C09106=1065.151,284.047,405.549,173.667,32.437,155.965
C09107=1065.146,283.799,405.580,173.664,32.433,155.964
C09108=1065.139,283.550,405.610,173.661,32.429,155.964
C09109=1065.133,283.302,405.641,173.659,32.425,155.963
C09110=1065.128,283.055,405.671,173.656,32.421,155.962
C09111=1065.121,282.806,405.702,173.653,32.416,155.961
C09112=1065.115,282.558,405.731,173.651,32.413,155.961
C09113=1065.109,282.311,405.762,173.648,32.409,155.960
C09114=1065.102,282.062,405.792,173.645,32.405,155.959
C09115=1065.097,281.814,405.823,173.642,32.401,155.958
C09116=1065.091,281.566,405.853,173.639,32.396,155.958
C09117=1065.084,281.318,405.884,173.637,32.393,155.957
C09118=1065.079,281.070,405.914,173.634,32.388,155.956
C09119=1065.073,280.822,405.945,173.631,32.384,155.955
C09120=1065.066,280.574,405.975,173.628,32.380,155.955
C09121=1065.060,280.326,406.006,173.625,32.376,155.954
C09122=1065.055,280.078,406.036,173.623,32.372,155.953
C09123=1065.048,279.829,406.065,173.621,32.368,155.952
C09124=1065.042,279.582,406.096,173.618,32.364,155.952
C09125=1065.036,279.334,406.126,173.615,32.360,155.951
C09126=1065.030,279.085,406.157,173.612,32.356,155.950
C09127=1065.023,278.838,406.187,173.609,32.352,155.949
C09128=1065.018,278.589,406.216,173.607,32.348,155.949
C09129=1065.011,278.341,406.247,173.604,32.344,155.948
C09130=1065.005,278.093,406.277,173.601,32.340,155.947
C09131=1064.999,277.845,406.306,173.598,32.336,155.946
C09132=1064.993,277.597,406.337,173.595,32.332,155.946
C09133=1064.987,277.377,406.364,173.594,32.328,155.945
C09134=1064.982,277.156,406.390,173.591,32.325,155.944
C09135=1064.976,276.936,406.417,173.589,32.321,155.944
C09136=1064.971,276.716,406.443,173.586,32.318,155.943
C09137=1064.966,276.496,406.470,173.584,32.314,155.942
C09138=1064.960,276.275,406.496,173.582,32.310,155.942
C09139=1064.955,276.055,406.524,173.579,32.307,155.941
C09140=1064.950,275.835,406.550,173.577,32.304,155.940
C09141=1064.943,275.587,406.580,173.574,32.299,155.940
C09142=1064.937,275.339,406.610,173.571,32.296,155.939
C09143=1064.932,275.091,406.640,173.568,32.291,155.938
C09144=1064.925,274.843,406.669,173.566,32.288,155.937
C09145=1064.920,274.595,406.699,173.564,32.283,155.937
C09146=1064.913,274.346,406.730,173.561,32.280,155.936
C09147=1064.907,274.098,406.759,173.558,32.275,155.935
C09148=1064.901,273.850,406.789,173.555,32.272,155.934
C09149=1064.895,273.602,406.818,173.553,32.267,155.934
C09150=1064.889,273.354,406.849,173.550,32.264,155.933
C09151=1064.883,273.106,406.878,173.547,32.259,155.932
C09152=1064.876,272.857,406.908,173.545,32.256,155.932
C09153=1064.870,272.609,406.937,173.542,32.251,155.931
C09154=1064.865,272.361,406.967,173.539,32.248,155.930
C09155=1064.858,272.113,406.997,173.537,32.243,155.929
C09156=1064.853,271.865,407.026,173.535,32.240,155.929
C09157=1064.846,271.617,407.055,173.532,32.235,155.928
C09158=1064.840,271.368,407.086,173.529,32.232,155.927
C09159=1064.834,271.120,407.115,173.526,32.227,155.926
C09160=1064.828,270.872,407.145,173.524,32.224,155.926
C09161=1064.822,270.624,407.175,173.521,32.219,155.925
C09162=1064.816,270.376,407.204,173.518,32.216,155.924
C09163=1064.810,270.128,407.233,173.515,32.211,155.923
C09164=1064.804,269.879,407.262,173.513,32.208,155.923
C09165=1064.798,269.632,407.293,173.511,32.204,155.922
C09166=1064.792,269.384,407.322,173.508,32.200,155.921
C09167=1064.786,269.135,407.351,173.506,32.196,155.921
C09168=1064.779,268.886,407.381,173.503,32.192,155.920
C09169=1064.773,268.639,407.410,173.500,32.188,155.919
C09170=1064.767,268.390,407.440,173.497,32.184,155.918
C09171=1064.761,268.142,407.469,173.495,32.180,155.918
C09172=1064.755,267.894,407.498,173.492,32.176,155.917
C09173=1064.749,267.646,407.528,173.489,32.172,155.916
C09174=1064.743,267.397,407.557,173.488,32.168,155.915
C09175=1064.737,267.149,407.586,173.485,32.164,155.915
C09176=1064.730,266.901,407.615,173.482,32.160,155.914
C09177=1064.725,266.653,407.645,173.480,32.156,155.913
C09178=1064.719,266.405,407.674,173.477,32.152,155.912
C09179=1064.712,266.157,407.703,173.474,32.148,155.912
C09180=1064.706,265.909,407.733,173.472,32.144,155.911
C09181=1064.700,265.661,407.762,173.469,32.140,155.910
C09182=1064.694,265.412,407.791,173.466,32.136,155.910
C09183=1064.688,265.164,407.820,173.465,32.133,155.909
C09184=1064.682,264.916,407.850,173.462,32.128,155.908
C09185=1064.676,264.667,407.878,173.459,32.124,155.907
C09186=1064.670,264.419,407.907,173.457,32.120,155.907
C09187=1064.664,264.171,407.936,173.454,32.116,155.906
C09188=1064.658,263.922,407.966,173.451,32.113,155.905
C09189=1064.653,263.704,407.991,173.449,32.109,155.905
C09190=1064.647,263.486,408.017,173.447,32.105,155.904
C09191=1064.642,263.268,408.042,173.444,32.102,155.903
C09192=1064.636,263.049,408.068,173.443,32.099,155.903
C09193=1064.631,262.831,408.093,173.440,32.095,155.902
C09194=1064.625,262.612,408.119,173.438,32.092,155.901
C09195=1064.619,262.393,408.144,173.436,32.089,155.901
C09196=1064.614,262.175,408.170,173.433,32.085,155.900
C09197=1064.608,261.927,408.199,173.431,32.081,155.899
C09198=1064.602,261.678,408.227,173.428,32.077,155.899
C09199=1064.595,261.430,408.256,173.425,32.073,155.898
C09200=1064.589,261.182,408.285,173.423,32.069,155.897
C09201=1064.583,260.934,408.314,173.421,32.066,155.897
C09202=1064.577,260.685,408.342,173.419,32.061,155.896
C09203=1064.571,260.437,408.371,173.416,32.058,155.895
C09204=1064.564,260.189,408.400,173.413,32.054,155.895
C09205=1064.558,259.940,408.429,173.411,32.050,155.894
C09206=1064.552,259.693,408.457,173.408,32.046,155.893
C09207=1064.546,259.445,408.486,173.405,32.042,155.892
C09208=1064.540,259.196,408.514,173.403,32.039,155.892
C09209=1064.534,258.948,408.543,173.401,32.034,155.891
C09210=1064.527,258.700,408.572,173.399,32.031,155.890
C09211=1064.521,258.451,408.601,173.396,32.027,155.890
C09212=1064.515,258.203,408.630,173.393,32.022,155.889
C09213=1064.509,257.954,408.658,173.391,32.019,155.888
C09214=1064.503,257.706,408.687,173.388,32.015,155.887
C09215=1064.496,257.458,408.715,173.385,32.011,155.887
C09216=1064.490,257.209,408.744,173.383,32.007,155.886
C09217=1064.485,256.961,408.772,173.381,32.003,155.885
C09218=1064.478,256.713,408.801,173.379,31.999,155.884
C09219=1064.473,256.464,408.829,173.376,31.995,155.884
C09220=1064.466,256.216,408.858,173.373,31.991,155.883
C09221=1064.460,255.968,408.886,173.371,31.987,155.882
C09222=1064.453,255.720,408.915,173.368,31.983,155.882
C09223=1064.448,255.472,408.943,173.366,31.979,155.881
C09224=1064.442,255.224,408.972,173.364,31.975,155.880
C09225=1064.436,254.975,409.000,173.362,31.972,155.880
C09226=1064.430,254.727,409.029,173.359,31.967,155.879
C09227=1064.424,254.478,409.058,173.356,31.964,155.878
C09228=1064.418,254.230,409.086,173.354,31.960,155.877
C09229=1064.411,253.982,409.114,173.351,31.956,155.877
C09230=1064.405,253.733,409.142,173.349,31.952,155.876
C09231=1064.399,253.485,409.171,173.347,31.948,155.875
C09232=1064.394,253.237,409.199,173.345,31.944,155.874
C09233=1064.388,252.988,409.228,173.342,31.940,155.874
C09234=1064.381,252.740,409.255,173.339,31.936,155.873
C09235=1064.375,252.492,409.284,173.337,31.932,155.872
C09236=1064.370,252.244,409.312,173.334,31.928,155.872
C09237=1064.364,251.995,409.341,173.332,31.924,155.871
C09238=1064.358,251.746,409.369,173.329,31.920,155.870
C09239=1064.351,251.498,409.397,173.328,31.916,155.869
C09240=1064.345,251.250,409.425,173.325,31.912,155.869
C09241=1064.339,251.002,409.454,173.323,31.908,155.868
C09242=1064.333,250.753,409.482,173.320,31.904,155.867
C09243=1064.328,250.505,409.510,173.318,31.901,155.867
C09244=1064.321,250.257,409.538,173.315,31.896,155.866
C09245=1064.316,250.037,409.564,173.313,31.893,155.865
C09246=1064.311,249.818,409.588,173.312,31.889,155.865
C09247=1064.305,249.598,409.613,173.309,31.886,155.864
C09248=1064.300,249.379,409.638,173.307,31.882,155.863
C09249=1064.295,249.159,409.663,173.305,31.879,155.863
C09250=1064.290,248.940,409.688,173.303,31.875,155.862
C09251=1064.285,248.720,409.713,173.300,31.871,155.861
C09252=1064.279,248.501,409.737,173.298,31.868,155.861
C09253=1064.273,248.252,409.766,173.297,31.864,155.860
C09254=1064.268,248.004,409.794,173.294,31.860,155.859
C09255=1064.261,247.755,409.821,173.292,31.856,155.858
C09256=1064.256,247.507,409.850,173.289,31.852,155.858
C09257=1064.250,247.259,409.878,173.287,31.848,155.857
C09258=1064.244,247.010,409.906,173.284,31.844,155.856
C09259=1064.238,246.762,409.933,173.282,31.840,155.856
C09260=1064.232,246.513,409.962,173.280,31.836,155.855
C09261=1064.227,246.265,409.990,173.278,31.832,155.854
C09262=1064.220,246.017,410.017,173.275,31.828,155.853
C09263=1064.214,245.768,410.046,173.273,31.824,155.853
C09264=1064.208,245.520,410.073,173.270,31.820,155.852
C09265=1064.202,245.272,410.101,173.268,31.816,155.851
C09266=1064.196,245.023,410.128,173.266,31.812,155.850
C09267=1064.190,244.775,410.156,173.264,31.808,155.850
C09268=1064.184,244.526,410.184,173.261,31.805,155.849
C09269=1064.178,244.278,410.212,173.259,31.800,155.848
C09270=1064.172,244.030,410.240,173.256,31.797,155.848
C09271=1064.166,243.782,410.268,173.254,31.792,155.847
C09272=1064.160,243.532,410.295,173.252,31.788,155.846
C09273=1064.154,243.284,410.323,173.250,31.785,155.846
C09274=1064.148,243.036,410.350,173.248,31.781,155.845
C09275=1064.142,242.787,410.379,173.245,31.777,155.844
C09276=1064.136,242.540,410.406,173.243,31.773,155.843
C09277=1064.130,242.290,410.434,173.240,31.769,155.843
C09278=1064.124,242.042,410.461,173.238,31.765,155.842
C09279=1064.118,241.794,410.489,173.236,31.761,155.841
C09280=1064.113,241.545,410.516,173.234,31.757,155.841
C09281=1064.106,241.297,410.544,173.231,31.753,155.840
C09282=1064.099,241.048,410.571,173.229,31.749,155.839
C09283=1064.094,240.800,410.599,173.226,31.745,155.838
C09284=1064.088,240.551,410.626,173.224,31.741,155.838
C09285=1064.081,240.304,410.654,173.223,31.737,155.837
C09286=1064.075,240.054,410.681,173.220,31.733,155.836
C09287=1064.070,239.806,410.709,173.218,31.730,155.836
C09288=1064.063,239.557,410.736,173.215,31.725,155.835
C09289=1064.057,239.310,410.763,173.213,31.722,155.834
C09290=1064.051,239.061,410.791,173.210,31.718,155.833
C09291=1064.046,238.813,410.818,173.209,31.714,155.833
C09292=1064.039,238.564,410.846,173.206,31.710,155.832
C09293=1064.033,238.316,410.873,173.204,31.705,155.831
C09294=1064.026,238.067,410.900,173.202,31.702,155.831
C09295=1064.021,237.819,410.928,173.199,31.698,155.830
C09296=1064.015,237.570,410.955,173.197,31.694,155.829
C09297=1064.009,237.322,410.982,173.195,31.690,155.828
C09298=1064.002,237.073,411.010,173.193,31.686,155.828
C09299=1063.996,236.825,411.036,173.190,31.682,155.827
C09300=1063.991,236.576,411.064,173.188,31.678,155.826
C09301=1063.985,236.354,411.088,173.186,31.674,155.826
C09302=1063.980,236.131,411.112,173.184,31.671,155.825
C09303=1063.975,235.909,411.137,173.183,31.668,155.824
C09304=1063.969,235.686,411.161,173.180,31.664,155.824
C09305=1063.964,235.463,411.186,173.178,31.660,155.823
C09306=1063.958,235.241,411.210,173.176,31.656,155.822
C09307=1063.953,235.018,411.234,173.174,31.653,155.822
C09308=1063.947,234.795,411.258,173.172,31.650,155.821
C09309=1063.941,234.547,411.286,173.170,31.646,155.820
C09310=1063.936,234.299,411.312,173.168,31.642,155.820
C09311=1063.929,234.049,411.339,173.166,31.638,155.819
C09312=1063.924,233.801,411.367,173.163,31.633,155.818
C09313=1063.918,233.553,411.394,173.161,31.630,155.818
C09314=1063.912,233.304,411.421,173.159,31.626,155.817
C09315=1063.906,233.056,411.448,173.157,31.622,155.816
C09316=1063.899,232.807,411.475,173.155,31.618,155.815
C09317=1063.893,232.559,411.502,173.152,31.614,155.815
C09318=1063.888,232.310,411.529,173.150,31.610,155.814
C09319=1063.881,232.061,411.556,173.148,31.606,155.813
C09320=1063.876,231.813,411.582,173.146,31.602,155.813
C09321=1063.869,231.565,411.610,173.144,31.598,155.812
C09322=1063.863,231.316,411.637,173.142,31.594,155.811
C09323=1063.857,231.068,411.663,173.139,31.590,155.810
C09324=1063.852,230.820,411.690,173.137,31.586,155.810
C09325=1063.845,230.570,411.717,173.135,31.582,155.809
C09326=1063.839,230.322,411.744,173.133,31.578,155.808
C09327=1063.833,230.074,411.771,173.131,31.574,155.807
C09328=1063.827,229.825,411.798,173.128,31.570,155.807
C09329=1063.821,229.577,411.825,173.126,31.566,155.806
C09330=1063.815,229.329,411.851,173.124,31.562,155.805
C09331=1063.809,229.080,411.878,173.122,31.558,155.805
C09332=1063.803,228.831,411.905,173.120,31.554,155.804
C09333=1063.797,228.583,411.932,173.118,31.550,155.803
C09334=1063.790,228.334,411.958,173.115,31.546,155.802
C09335=1063.785,228.086,411.985,173.113,31.542,155.802
C09336=1063.779,227.837,412.011,173.112,31.538,155.801
C09337=1063.773,227.589,412.038,173.109,31.534,155.800
C09338=1063.767,227.340,412.065,173.107,31.530,155.800
C09339=1063.760,227.092,412.091,173.105,31.526,155.799
C09340=1063.754,226.844,412.118,173.102,31.522,155.798
C09341=1063.748,226.594,412.144,173.101,31.518,155.797
C09342=1063.743,226.345,412.171,173.099,31.514,155.797
C09343=1063.737,226.097,412.197,173.096,31.510,155.796
C09344=1063.730,225.849,412.223,173.094,31.506,155.795
C09345=1063.724,225.600,412.251,173.092,31.503,155.795
C09346=1063.718,225.352,412.277,173.090,31.498,155.794
C09347=1063.712,225.103,412.304,173.088,31.494,155.793
C09348=1063.706,224.855,412.330,173.086,31.490,155.792
C09349=1063.700,224.606,412.356,173.083,31.486,155.792
C09350=1063.694,224.357,412.383,173.081,31.483,155.791
C09351=1063.688,224.109,412.409,173.080,31.478,155.790
C09352=1063.682,223.861,412.436,173.077,31.474,155.790
C09353=1063.676,223.612,412.462,173.075,31.470,155.789
C09354=1063.670,223.363,412.488,173.073,31.466,155.788
C09355=1063.664,223.114,412.515,173.071,31.462,155.787
C09356=1063.658,222.866,412.541,173.069,31.458,155.787
C09357=1063.652,222.640,412.565,173.067,31.455,155.786
C09358=1063.647,222.413,412.589,173.065,31.451,155.785
C09359=1063.642,222.186,412.614,173.063,31.447,155.785
C09360=1063.636,221.960,412.638,173.061,31.444,155.784
C09361=1063.631,221.733,412.662,173.059,31.440,155.783
C09362=1063.625,221.507,412.685,173.058,31.436,155.783
C09363=1063.620,221.280,412.709,173.056,31.432,155.782
C09364=1063.614,221.053,412.733,173.054,31.429,155.781
C09365=1063.608,220.805,412.759,173.051,31.425,155.781
C09366=1063.602,220.556,412.785,173.049,31.421,155.780
C09367=1063.597,220.308,412.812,173.048,31.417,155.779
C09368=1063.590,220.058,412.838,173.045,31.413,155.779
C09369=1063.584,219.810,412.864,173.043,31.409,155.778
C09370=1063.578,219.562,412.890,173.041,31.405,155.777
C09371=1063.572,219.313,412.916,173.040,31.401,155.776
C09372=1063.566,219.065,412.942,173.037,31.397,155.776
C09373=1063.560,218.816,412.968,173.035,31.393,155.775
C09374=1063.554,218.568,412.994,173.033,31.389,155.774
C09375=1063.548,218.319,413.020,173.031,31.385,155.773
C09376=1063.541,218.070,413.047,173.029,31.381,155.773
C09377=1063.536,217.821,413.073,173.027,31.377,155.772
C09378=1063.529,217.573,413.099,173.025,31.373,155.771
C09379=1063.523,217.324,413.124,173.023,31.369,155.771
C09380=1063.517,217.076,413.151,173.020,31.365,155.770
C09381=1063.511,216.827,413.176,173.019,31.361,155.769
C09382=1063.505,216.579,413.203,173.017,31.357,155.768
C09383=1063.499,216.330,413.228,173.015,31.353,155.768
C09384=1063.493,216.081,413.254,173.012,31.348,155.767
C09385=1063.487,215.833,413.280,173.011,31.345,155.766
C09386=1063.481,215.584,413.306,173.009,31.340,155.766
C09387=1063.475,215.336,413.332,173.007,31.337,155.765
C09388=1063.469,215.087,413.358,173.004,31.332,155.764
C09389=1063.463,214.839,413.383,173.002,31.328,155.763
C09390=1063.457,214.590,413.410,173.001,31.324,155.763
C09391=1063.451,214.342,413.435,172.999,31.320,155.762
C09392=1063.445,214.093,413.461,172.996,31.316,155.761
C09393=1063.439,213.845,413.487,172.994,31.312,155.760
C09394=1063.433,213.596,413.513,172.993,31.308,155.760
C09395=1063.428,213.347,413.539,172.991,31.304,155.759
C09396=1063.421,213.099,413.565,172.989,31.300,155.758
C09397=1063.416,212.850,413.591,172.986,31.296,155.757
C09398=1063.409,212.601,413.616,172.984,31.291,155.757
C09399=1063.403,212.352,413.641,172.983,31.288,155.756
C09400=1063.397,212.104,413.668,172.981,31.283,155.755
C09401=1063.391,211.855,413.693,172.979,31.280,155.755
C09402=1063.385,211.607,413.719,172.976,31.275,155.754
C09403=1063.379,211.358,413.744,172.975,31.271,155.753
C09404=1063.373,211.109,413.770,172.973,31.267,155.752
C09405=1063.367,210.860,413.795,172.971,31.263,155.752
C09406=1063.361,210.612,413.821,172.969,31.259,155.751
C09407=1063.354,210.364,413.847,172.967,31.255,155.750
C09408=1063.349,210.115,413.872,172.965,31.251,155.749
C09409=1063.343,209.866,413.898,172.963,31.247,155.749
C09410=1063.337,209.617,413.923,172.961,31.243,155.748
C09411=1063.330,209.369,413.949,172.959,31.239,155.747
C09412=1063.325,209.120,413.974,172.957,31.235,155.747
C09413=1063.319,208.896,413.997,172.955,31.231,155.746
C09414=1063.314,208.672,414.020,172.953,31.227,155.745
C09415=1063.308,208.448,414.044,172.951,31.224,155.745
C09416=1063.302,208.223,414.066,172.950,31.220,155.744
C09417=1063.298,207.999,414.089,172.949,31.216,155.743
C09418=1063.292,207.775,414.112,172.947,31.213,155.743
C09419=1063.286,207.551,414.135,172.945,31.209,155.742
C09420=1063.281,207.326,414.158,172.943,31.205,155.741
C09421=1063.256,206.279,414.261,172.776,31.124,155.734
C09422=1063.250,206.030,414.286,172.774,31.121,155.734
C09423=1063.245,205.781,414.310,172.771,31.118,155.733
C09424=1063.238,205.533,414.335,172.769,31.114,155.733
C09425=1063.233,205.284,414.359,172.766,31.111,155.732
C09426=1063.227,205.035,414.384,172.765,31.108,155.732
C09427=1063.222,204.787,414.408,172.763,31.105,155.731
C09428=1063.216,204.538,414.434,172.760,31.102,155.731
C09429=1063.210,204.289,414.458,172.758,31.099,155.730
C09430=1063.204,204.040,414.482,172.755,31.095,155.730
C09431=1063.198,203.792,414.506,172.754,31.092,155.729
C09432=1063.192,203.542,414.531,172.751,31.089,155.729
C09433=1063.187,203.294,414.556,172.749,31.086,155.728
C09434=1063.181,203.045,414.580,172.746,31.082,155.727
C09435=1063.176,202.797,414.605,172.744,31.079,155.727
C09436=1063.169,202.548,414.629,172.743,31.076,155.726
C09437=1063.164,202.299,414.653,172.740,31.073,155.726
C09438=1063.158,202.050,414.677,172.738,31.070,155.725
C09439=1063.152,201.801,414.701,172.735,31.067,155.725
C09440=1063.146,201.554,414.726,172.734,31.063,155.724
C09441=1063.140,201.304,414.751,172.731,31.061,155.724
C09442=1063.134,201.056,414.774,172.729,31.057,155.723
C09443=1063.128,200.807,414.799,172.727,31.054,155.723
C09444=1063.122,200.558,414.823,172.724,31.051,155.722
C09445=1063.116,200.309,414.847,172.723,31.048,155.722
C09446=1063.110,200.061,414.871,172.720,31.045,155.721
C09447=1063.104,199.812,414.896,172.718,31.042,155.721
C09448=1063.098,199.563,414.919,172.715,31.039,155.720
C09449=1063.092,199.314,414.944,172.713,31.036,155.720
C09450=1063.086,199.066,414.968,172.712,31.033,155.719
C09451=1063.081,198.817,414.992,172.709,31.030,155.719
C09452=1063.075,198.568,415.016,172.707,31.027,155.718
C09453=1063.070,198.319,415.039,172.704,31.023,155.718
C09454=1063.063,198.070,415.063,172.702,31.020,155.717
C09455=1063.058,197.821,415.088,172.701,31.017,155.717
C09456=1063.051,197.572,415.112,172.698,31.014,155.716
C09457=1063.046,197.324,415.136,172.696,31.011,155.716
C09458=1063.040,197.075,415.160,172.693,31.008,155.715
C09459=1063.034,196.826,415.184,172.692,31.005,155.715
C09460=1063.028,196.578,415.208,172.690,31.002,155.714
C09461=1063.022,196.329,415.232,172.687,30.999,155.714
C09462=1063.016,196.080,415.255,172.685,30.996,155.713
C09463=1063.011,195.831,415.280,172.682,30.992,155.713
C09464=1063.005,195.583,415.303,172.681,30.990,155.713
C09465=1062.999,195.334,415.328,172.679,30.987,155.712
C09466=1062.993,195.085,415.352,172.676,30.983,155.711
C09467=1062.988,194.836,415.375,172.674,30.981,155.711
C09468=1062.981,194.587,415.399,172.672,30.977,155.710
C09469=1062.975,194.339,415.423,172.670,30.974,155.710
C09470=1062.970,194.090,415.447,172.668,30.971,155.710
C09471=1062.963,193.841,415.470,172.666,30.968,155.709
C09472=1062.958,193.592,415.495,172.663,30.965,155.708
C09473=1062.952,193.344,415.518,172.662,30.962,155.708
C09474=1062.946,193.095,415.543,172.659,30.959,155.708
C09475=1062.940,192.846,415.566,172.657,30.956,155.707
C09476=1062.935,192.597,415.590,172.655,30.953,155.707
C09477=1062.929,192.349,415.614,172.652,30.950,155.706
C09478=1062.923,192.099,415.637,172.651,30.947,155.706
C09479=1062.918,191.851,415.661,172.649,30.944,155.705
C09480=1062.911,191.602,415.685,172.646,30.941,155.705
C09481=1062.907,191.353,415.709,172.644,30.937,155.704
C09482=1062.899,191.070,415.736,172.642,30.934,155.704
C09483=1062.893,190.786,415.762,172.640,30.931,155.703
C09484=1062.887,190.504,415.790,172.637,30.927,155.702
C09485=1062.879,190.220,415.817,172.634,30.924,155.702
C09486=1062.874,189.971,415.840,172.633,30.920,155.701
C09487=1062.868,189.723,415.864,172.631,30.918,155.701
C09488=1062.863,189.474,415.887,172.629,30.914,155.700
C09489=1062.857,189.225,415.912,172.626,30.911,155.700
C09490=1062.851,188.976,415.934,172.624,30.908,155.699
C09491=1062.846,188.727,415.959,172.623,30.905,155.699
C09492=1062.840,188.478,415.982,172.620,30.902,155.698
C09493=1062.834,188.230,416.005,172.618,30.899,155.698
C09494=1062.829,187.981,416.029,172.616,30.896,155.697
C09495=1062.822,187.732,416.053,172.613,30.893,155.697
C09496=1062.817,187.483,416.076,172.612,30.890,155.696
C09497=1062.811,187.234,416.100,172.610,30.887,155.696
C09498=1062.806,186.986,416.123,172.608,30.884,155.695
C09499=1062.800,186.737,416.147,172.605,30.881,155.695
C09500=1062.795,186.488,416.170,172.604,30.878,155.694
C09501=1062.789,186.240,416.194,172.602,30.875,155.694
C09502=1062.784,185.991,416.217,172.599,30.872,155.694
C09503=1062.778,185.742,416.240,172.597,30.868,155.693
C09504=1062.771,185.493,416.264,172.595,30.866,155.693
C09505=1062.766,185.244,416.288,172.594,30.863,155.692
C09506=1062.760,184.995,416.312,172.591,30.859,155.691
C09507=1062.755,184.746,416.335,172.589,30.857,155.691
C09508=1062.749,184.497,416.358,172.587,30.853,155.691
C09509=1062.744,184.248,416.381,172.585,30.851,155.690
C09510=1062.738,184.000,416.405,172.583,30.847,155.690
C09511=1062.731,183.750,416.428,172.581,30.845,155.689
C09512=1062.725,183.502,416.450,172.579,30.842,155.689
C09513=1062.719,183.253,416.473,172.577,30.839,155.688
C09514=1062.713,183.005,416.497,172.575,30.836,155.688
C09515=1062.707,182.756,416.520,172.573,30.834,155.687
C09516=1062.701,182.506,416.543,172.570,30.830,155.687
C09517=1062.695,182.257,416.566,172.568,30.827,155.686
C09518=1062.690,182.008,416.589,172.567,30.825,155.686
C09519=1062.684,181.760,416.613,172.565,30.822,155.686
C09520=1062.678,181.511,416.636,172.562,30.819,155.685
C09521=1062.671,181.263,416.658,172.560,30.816,155.685
C09522=1062.665,181.013,416.681,172.558,30.813,155.684
C09523=1062.659,180.764,416.704,172.557,30.810,155.684
C09524=1062.654,180.515,416.727,172.554,30.808,155.683
C09525=1062.648,180.266,416.750,172.552,30.804,155.683
C09526=1062.642,180.018,416.774,172.550,30.802,155.682
C09527=1062.636,179.769,416.797,172.549,30.798,155.682
C09528=1062.630,179.520,416.820,172.546,30.796,155.681
C09529=1062.624,179.272,416.842,172.544,30.793,155.681
C09530=1062.618,179.023,416.865,172.542,30.790,155.680
C09531=1062.612,178.773,416.888,172.540,30.787,155.680
C09532=1062.606,178.524,416.911,172.538,30.784,155.680
C09533=1062.600,178.275,416.934,172.536,30.781,155.679
C09534=1062.595,178.026,416.957,172.534,30.779,155.679
C09535=1062.588,177.778,416.980,172.532,30.776,155.678
C09536=1062.582,177.529,417.003,172.530,30.772,155.678
C09537=1062.577,177.280,417.026,172.528,30.770,155.677
C09538=1062.571,177.031,417.048,172.526,30.767,155.677
C09539=1062.565,176.782,417.071,172.524,30.764,155.676
C09540=1062.559,176.533,417.094,172.521,30.761,155.676
C09541=1062.553,176.285,417.117,172.520,30.759,155.676
C09542=1062.547,176.036,417.140,172.518,30.755,155.675
C09543=1062.542,175.787,417.163,172.516,30.753,155.675
C09544=1062.536,175.538,417.186,172.514,30.749,155.674
C09545=1062.530,175.289,417.208,172.512,30.747,155.674
C09546=1062.524,175.005,417.234,172.510,30.743,155.673
C09547=1062.517,174.722,417.260,172.507,30.740,155.673
C09548=1062.510,174.439,417.286,172.505,30.737,155.672
C09549=1062.504,174.155,417.312,172.503,30.733,155.672
C09550=1062.498,173.906,417.334,172.501,30.731,155.671
C09551=1062.492,173.657,417.357,172.499,30.728,155.671
C09552=1062.486,173.408,417.380,172.497,30.725,155.670
C09553=1062.480,173.159,417.403,172.495,30.722,155.670
C09554=1062.475,172.910,417.425,172.493,30.719,155.669
C09555=1062.468,172.661,417.447,172.491,30.716,155.669
C09556=1062.462,172.412,417.470,172.489,30.714,155.668
C09557=1062.457,172.164,417.493,172.487,30.710,155.668
C09558=1062.451,171.915,417.516,172.486,30.708,155.668
C09559=1062.446,171.665,417.538,172.483,30.705,155.667
C09560=1062.439,171.417,417.561,172.481,30.702,155.667
C09561=1062.433,171.168,417.584,172.479,30.699,155.666
C09562=1062.428,170.919,417.607,172.478,30.696,155.666
C09563=1062.423,170.670,417.628,172.476,30.693,155.665
C09564=1062.416,170.421,417.651,172.474,30.691,155.665
C09565=1062.411,170.173,417.674,172.471,30.688,155.664
C09566=1062.405,169.924,417.697,172.469,30.684,155.664
C09567=1062.399,169.674,417.719,172.468,30.682,155.663
C09568=1062.393,169.426,417.741,172.466,30.679,155.663
C09569=1062.387,169.177,417.764,172.464,30.676,155.662
C09570=1062.382,168.928,417.786,172.462,30.673,155.662
C09571=1062.377,168.679,417.809,172.460,30.670,155.662
C09572=1062.370,168.430,417.831,172.458,30.667,155.661
C09573=1062.365,168.181,417.854,172.456,30.665,155.661
C09574=1062.359,167.932,417.877,172.454,30.661,155.660
C09575=1062.353,167.683,417.898,172.453,30.659,155.660
C09576=1062.348,167.435,417.921,172.451,30.656,155.659
C09577=1062.342,167.186,417.944,172.449,30.653,155.659
C09578=1062.337,166.936,417.966,172.446,30.650,155.658
C09579=1062.330,166.688,417.988,172.444,30.647,155.658
C09580=1062.325,166.438,418.011,172.443,30.644,155.657
C09581=1062.320,166.190,418.033,172.441,30.642,155.657
C09582=1062.313,165.941,418.055,172.439,30.638,155.657
C09583=1062.308,165.692,418.078,172.437,30.636,155.656
C09584=1062.302,165.443,418.101,172.436,30.633,155.656
C09585=1062.297,165.193,418.123,172.434,30.630,155.655
C09586=1062.291,164.945,418.145,172.431,30.627,155.655
C09587=1062.285,164.696,418.167,172.429,30.624,155.654
C09588=1062.280,164.447,418.190,172.428,30.621,155.654
C09589=1062.273,164.198,418.212,172.426,30.618,155.653
C09590=1062.268,163.950,418.234,172.424,30.615,155.653
C09591=1062.263,163.700,418.256,172.422,30.612,155.652
C09592=1062.257,163.451,418.278,172.420,30.610,155.652
C09593=1062.251,163.202,418.301,172.419,30.607,155.652
C09594=1062.246,162.953,418.323,172.417,30.604,155.651
C09595=1062.240,162.705,418.345,172.414,30.601,155.651
C09596=1062.234,162.455,418.368,172.412,30.598,155.650
C09597=1062.229,162.207,418.390,172.411,30.595,155.650
C09598=1062.223,161.958,418.412,172.409,30.592,155.649
C09599=1062.217,161.708,418.434,172.407,30.589,155.649
C09600=1062.212,161.460,418.457,172.405,30.586,155.648
C09601=1062.206,161.211,418.478,172.404,30.583,155.648
C09602=1062.201,160.961,418.500,172.402,30.581,155.647
C09603=1062.194,160.713,418.523,172.400,30.578,155.647
C09604=1062.189,160.464,418.544,172.398,30.575,155.646
C09605=1062.183,160.215,418.566,172.396,30.572,155.646
C09606=1062.177,159.966,418.589,172.394,30.569,155.646
C09607=1062.171,159.717,418.610,172.392,30.567,155.645
C09608=1062.166,159.468,418.632,172.390,30.564,155.645
C09609=1062.160,159.219,418.654,172.388,30.561,155.644
C09610=1062.153,158.935,418.679,172.387,30.558,155.644
C09611=1062.146,158.651,418.704,172.384,30.555,155.643
C09612=1062.140,158.367,418.729,172.382,30.552,155.643
C09613=1062.133,158.083,418.753,172.381,30.548,155.642
C09614=1062.127,157.834,418.776,172.378,30.545,155.642
C09615=1062.121,157.585,418.798,172.376,30.543,155.642
C09616=1062.115,157.337,418.819,172.374,30.540,155.641
C09617=1062.110,157.087,418.842,172.373,30.537,155.641
C09618=1062.104,156.838,418.863,172.371,30.534,155.640
C09619=1062.098,156.589,418.884,172.369,30.532,155.640
C09620=1062.092,156.340,418.907,172.367,30.529,155.639
C09621=1062.086,156.091,418.929,172.365,30.526,155.639
C09622=1062.081,155.843,418.950,172.364,30.523,155.638
C09623=1062.075,155.593,418.972,172.362,30.520,155.638
C09624=1062.069,155.344,418.994,172.360,30.518,155.638
C09625=1062.064,155.095,419.015,172.358,30.515,155.637
C09626=1062.057,154.846,419.037,172.357,30.512,155.637
C09627=1062.051,154.597,419.059,172.354,30.510,155.636
C09628=1062.046,154.349,419.080,172.352,30.506,155.636
C09629=1062.040,154.099,419.102,172.350,30.504,155.635
C09630=1062.034,153.850,419.124,172.349,30.501,155.635
C09631=1062.029,153.601,419.145,172.347,30.498,155.635
C09632=1062.022,153.352,419.167,172.345,30.496,155.634
C09633=1062.016,153.103,419.188,172.343,30.493,155.634
C09634=1062.010,152.855,419.210,172.342,30.490,155.633
C09635=1062.005,152.605,419.232,172.340,30.487,155.633
C09636=1061.999,152.356,419.254,172.338,30.484,155.632
C09637=1061.994,152.107,419.275,172.336,30.482,155.632
C09638=1061.987,151.858,419.296,172.334,30.479,155.632
C09639=1061.982,151.609,419.318,172.333,30.476,155.631
C09640=1061.976,151.360,419.339,172.331,30.474,155.631
C09641=1061.969,151.111,419.361,172.329,30.470,155.630
C09642=1061.964,150.863,419.382,172.327,30.468,155.630
C09643=1061.958,150.613,419.404,172.326,30.465,155.629
C09644=1061.953,150.365,419.426,172.324,30.462,155.629
C09645=1061.947,150.115,419.447,172.322,30.460,155.629
C09646=1061.941,149.866,419.469,172.320,30.457,155.628
C09647=1061.935,149.618,419.490,172.319,30.454,155.628
C09648=1061.929,149.368,419.512,172.317,30.451,155.627
C09649=1061.924,149.119,419.532,172.314,30.448,155.627
C09650=1061.917,148.870,419.554,172.312,30.446,155.626
C09651=1061.912,148.622,419.575,172.311,30.443,155.626
C09652=1061.906,148.372,419.597,172.309,30.440,155.626
C09653=1061.900,148.123,419.619,172.307,30.438,155.625
C09654=1061.894,147.875,419.640,172.305,30.434,155.625
C09655=1061.888,147.625,419.661,172.304,30.432,155.624
C09656=1061.883,147.376,419.682,172.302,30.429,155.624
C09657=1061.876,147.127,419.704,172.300,30.426,155.623
C09658=1061.871,146.879,419.725,172.298,30.424,155.623
C09659=1061.865,146.629,419.746,172.296,30.421,155.623
C09660=1061.859,146.380,419.768,172.295,30.418,155.622
C09661=1061.853,146.131,419.789,172.293,30.416,155.622
C09662=1061.847,145.882,419.810,172.291,30.413,155.621
C09663=1061.842,145.633,419.831,172.289,30.410,155.621
C09664=1061.835,145.384,419.852,172.288,30.408,155.620
C09665=1061.829,145.135,419.873,172.286,30.405,155.620
C09666=1061.824,144.886,419.894,172.284,30.402,155.620
C09667=1061.818,144.637,419.916,172.282,30.399,155.619
C09668=1061.812,144.388,419.937,172.281,30.396,155.619
C09669=1061.806,144.139,419.958,172.279,30.394,155.618
C09670=1061.800,143.889,419.979,172.277,30.391,155.618
C09671=1061.795,143.641,420.001,172.275,30.388,155.617
C09672=1061.789,143.391,420.022,172.274,30.386,155.617
C09673=1061.783,143.143,420.042,172.272,30.383,155.617
C09674=1061.777,142.859,420.067,172.270,30.380,155.616
C09675=1061.769,142.574,420.091,172.268,30.377,155.616
C09676=1061.763,142.290,420.115,172.266,30.374,155.615
C09677=1061.756,142.006,420.139,172.264,30.370,155.615
C09678=1061.751,141.757,420.160,172.262,30.368,155.614
C09679=1061.745,141.507,420.181,172.260,30.365,155.614
C09680=1061.739,141.258,420.202,172.259,30.362,155.613
C09681=1061.732,141.009,420.223,172.257,30.360,155.613
C09682=1061.727,140.760,420.244,172.255,30.357,155.613
C09683=1061.721,140.511,420.265,172.253,30.354,155.612
C09684=1061.715,140.263,420.286,172.252,30.351,155.612
C09685=1061.710,140.013,420.307,172.250,30.348,155.611
C09686=1061.703,139.765,420.328,172.248,30.346,155.611
C09687=1061.698,139.515,420.349,172.246,30.343,155.610
C09688=1061.692,139.266,420.369,172.245,30.340,155.610
C09689=1061.687,139.017,420.391,172.243,30.338,155.610
C09690=1061.680,138.768,420.411,172.241,30.335,155.609
C09691=1061.674,138.519,420.432,172.239,30.332,155.609
C09692=1061.669,138.270,420.453,172.238,30.330,155.608
C09693=1061.662,138.021,420.474,172.236,30.327,155.608
C09694=1061.657,137.772,420.494,172.234,30.324,155.608
C09695=1061.651,137.523,420.516,172.232,30.322,155.607
C09696=1061.645,137.274,420.536,172.232,30.319,155.607
C09697=1061.639,137.024,420.557,172.230,30.316,155.606
C09698=1061.633,136.776,420.578,172.228,30.314,155.606
C09699=1061.627,136.527,420.598,172.226,30.311,155.605
C09700=1061.622,136.277,420.619,172.225,30.308,155.605
C09701=1061.616,136.028,420.640,172.223,30.306,155.605
C09702=1061.609,135.779,420.661,172.221,30.302,155.604
C09703=1061.604,135.530,420.682,172.219,30.300,155.604
C09704=1061.598,135.282,420.702,172.218,30.297,155.603
C09705=1061.592,135.032,420.723,172.216,30.294,155.603
C09706=1061.587,134.783,420.743,172.214,30.292,155.602
C09707=1061.580,134.534,420.764,172.212,30.289,155.602
C09708=1061.575,134.285,420.785,172.211,30.286,155.602
C09709=1061.569,134.035,420.806,172.209,30.284,155.601
C09710=1061.562,133.787,420.827,172.207,30.281,155.601
C09711=1061.557,133.537,420.847,172.205,30.278,155.600
C09712=1061.551,133.289,420.867,172.204,30.276,155.600
C09713=1061.545,133.039,420.888,172.202,30.273,155.600
C09714=1061.540,132.790,420.909,172.200,30.270,155.599
C09715=1061.534,132.542,420.929,172.198,30.268,155.599
C09716=1061.528,132.292,420.950,172.197,30.265,155.598
C09717=1061.522,132.043,420.970,172.196,30.262,155.598
C09718=1061.516,131.794,420.991,172.194,30.260,155.598
C09719=1061.510,131.545,421.012,172.192,30.257,155.597
C09720=1061.504,131.296,421.032,172.190,30.254,155.597
C09721=1061.498,131.047,421.052,172.189,30.252,155.596
C09722=1061.492,130.797,421.073,172.187,30.249,155.596
C09723=1061.487,130.548,421.093,172.185,30.246,155.595
C09724=1061.480,130.299,421.113,172.183,30.244,155.595
C09725=1061.474,130.051,421.134,172.182,30.241,155.595
C09726=1061.468,129.801,421.155,172.180,30.238,155.594
C09727=1061.462,129.552,421.175,172.178,30.235,155.594
C09728=1061.456,129.303,421.195,172.176,30.233,155.593
C09729=1061.451,129.054,421.216,172.175,30.230,155.593
C09730=1061.444,128.804,421.236,172.173,30.227,155.593
C09731=1061.438,128.556,421.256,172.171,30.225,155.592
C09732=1061.433,128.307,421.276,172.169,30.223,155.592
C09733=1061.426,128.057,421.297,172.169,30.220,155.591
C09734=1061.420,127.808,421.317,172.167,30.217,155.591
C09735=1061.415,127.559,421.337,172.165,30.215,155.591
C09736=1061.408,127.310,421.358,172.163,30.212,155.590
C09737=1061.402,127.061,421.378,172.162,30.209,155.590
C09738=1061.396,126.777,421.402,172.160,30.206,155.589
C09739=1061.389,126.492,421.424,172.157,30.203,155.589
C09740=1061.382,126.208,421.447,172.156,30.200,155.588
C09741=1061.375,125.923,421.470,172.154,30.197,155.588
C09742=1061.369,125.675,421.490,172.152,30.195,155.588
C09743=1061.364,125.425,421.511,172.150,30.192,155.587
C09744=1061.358,125.177,421.531,172.149,30.189,155.587
C09745=1061.351,124.927,421.551,172.147,30.186,155.586
C09746=1061.346,124.678,421.572,172.146,30.184,155.586
C09747=1061.340,124.429,421.591,172.144,30.181,155.586
C09748=1061.334,124.180,421.611,172.143,30.179,155.585
C09749=1061.327,123.931,421.632,172.141,30.176,155.585
C09750=1061.322,123.681,421.652,172.139,30.173,155.584
C09751=1061.316,123.432,421.672,172.137,30.170,155.584
C09752=1061.310,123.183,421.692,172.136,30.168,155.583
C09753=1061.305,122.934,421.712,172.134,30.165,155.583
C09754=1061.298,122.685,421.732,172.132,30.162,155.583
C09755=1061.292,122.436,421.752,172.130,30.160,155.582
C09756=1061.286,122.187,421.772,172.129,30.157,155.582
C09757=1061.281,121.938,421.793,172.128,30.155,155.581
C09758=1061.276,121.689,421.812,172.126,30.152,155.581
C09759=1061.269,121.439,421.832,172.124,30.149,155.581
C09760=1061.263,121.190,421.852,172.123,30.146,155.580
C09761=1061.258,120.941,421.873,172.121,30.144,155.580
C09762=1061.252,120.692,421.893,172.119,30.141,155.579
C09763=1061.246,120.443,421.912,172.117,30.138,155.579
C09764=1061.240,120.194,421.932,172.116,30.136,155.579
C09765=1061.234,119.944,421.953,172.115,30.133,155.578
C09766=1061.228,119.695,421.973,172.113,30.130,155.578
C09767=1061.222,119.446,421.992,172.111,30.128,155.577
C09768=1061.217,119.197,422.012,172.110,30.125,155.577
C09769=1061.211,118.948,422.032,172.108,30.122,155.576
C09770=1061.205,118.699,422.053,172.106,30.120,155.576
C09771=1061.200,118.450,422.072,172.105,30.117,155.576
C09772=1061.194,118.201,422.092,172.103,30.114,155.575
C09773=1061.187,117.952,422.112,172.101,30.112,155.575
C09774=1061.182,117.702,422.133,172.100,30.109,155.574
C09775=1061.176,117.453,422.152,172.099,30.106,155.574
C09776=1061.170,117.204,422.172,172.097,30.104,155.574
C09777=1061.164,116.955,422.192,172.095,30.101,155.573
C09778=1061.158,116.706,422.211,172.093,30.098,155.573
C09779=1061.153,116.457,422.232,172.092,30.096,155.572
C09780=1061.147,116.208,422.252,172.090,30.093,155.572
C09781=1061.141,115.959,422.271,172.089,30.090,155.572
C09782=1061.135,115.710,422.291,172.087,30.088,155.571
C09783=1061.130,115.460,422.310,172.086,30.084,155.571
C09784=1061.124,115.211,422.331,172.084,30.082,155.570
C09785=1061.118,114.962,422.351,172.082,30.079,155.570
C09786=1061.112,114.712,422.370,172.080,30.076,155.569
C09787=1061.106,114.463,422.390,172.079,30.074,155.569
C09788=1061.101,114.214,422.409,172.078,30.071,155.569
C09789=1061.095,113.965,422.429,172.076,30.068,155.568
C09790=1061.089,113.716,422.449,172.074,30.066,155.568
C09791=1061.083,113.467,422.469,172.073,30.063,155.567
C09792=1061.077,113.218,422.489,172.071,30.060,155.567
C09793=1061.071,112.969,422.508,172.069,30.057,155.566
C09794=1061.065,112.720,422.528,172.068,30.055,155.566
C09795=1061.059,112.470,422.547,172.067,30.053,155.566
C09796=1061.053,112.222,422.567,172.065,30.050,155.565
C09797=1061.048,111.972,422.586,172.063,30.047,155.565
C09798=1061.042,111.723,422.606,172.062,30.045,155.565
C09799=1061.036,111.474,422.625,172.060,30.042,155.564
C09800=1061.030,111.224,422.645,172.058,30.039,155.564
C09801=1061.024,110.975,422.665,172.056,30.037,155.563
C09802=1061.018,110.691,422.687,172.055,30.033,155.563
C09803=1061.010,110.406,422.709,172.053,30.031,155.562
C09804=1061.004,110.121,422.731,172.051,30.028,155.562
C09805=1060.997,109.838,422.754,172.050,30.025,155.561
C09806=1060.990,109.588,422.773,172.048,30.022,155.561
C09807=1060.984,109.339,422.793,172.046,30.019,155.561
C09808=1060.978,109.090,422.812,172.044,30.016,155.560
C09809=1060.973,108.840,422.831,172.043,30.014,155.560
C09810=1060.967,108.591,422.851,172.042,30.012,155.560
C09811=1060.961,108.342,422.870,172.040,30.009,155.559
C09812=1060.955,108.093,422.889,172.038,30.006,155.559
C09813=1060.949,107.844,422.909,172.037,30.004,155.558
C09814=1060.943,107.595,422.928,172.035,30.001,155.558
C09815=1060.937,107.345,422.947,172.033,29.998,155.558
C09816=1060.931,107.096,422.967,172.032,29.996,155.557
C09817=1060.925,106.847,422.986,172.031,29.993,155.557
C09818=1060.919,106.598,423.005,172.029,29.990,155.556
C09819=1060.913,106.349,423.025,172.027,29.988,155.556
C09820=1060.907,106.100,423.044,172.025,29.986,155.556
C09821=1060.901,105.850,423.063,172.024,29.983,155.555
C09822=1060.895,105.601,423.082,172.022,29.980,155.555
C09823=1060.889,105.352,423.102,172.021,29.978,155.554
C09824=1060.884,105.103,423.122,172.020,29.975,155.554
C09825=1060.878,104.853,423.141,172.018,29.972,155.554
C09826=1060.871,104.604,423.159,172.016,29.969,155.553
C09827=1060.865,104.355,423.179,172.014,29.967,155.553
C09828=1060.860,104.107,423.198,172.013,29.964,155.552
C09829=1060.855,103.857,423.218,172.012,29.962,155.552
C09830=1060.848,103.608,423.236,172.010,29.959,155.551
C09831=1060.843,103.359,423.255,172.008,29.956,155.551
C09832=1060.837,103.110,423.275,172.007,29.953,155.551
C09833=1060.831,102.860,423.295,172.005,29.951,155.550
C09834=1060.824,102.611,423.313,172.004,29.948,155.550
C09835=1060.819,102.362,423.333,172.003,29.945,155.549
C09836=1060.813,102.112,423.352,172.001,29.943,155.549
C09837=1060.807,101.863,423.371,171.999,29.940,155.549
C09838=1060.801,101.614,423.390,171.997,29.937,155.548
C09839=1060.795,101.365,423.410,171.996,29.935,155.548
C09840=1060.790,101.116,423.428,171.995,29.933,155.547
C09841=1060.784,100.867,423.448,171.993,29.930,155.547
C09842=1060.778,100.618,423.466,171.991,29.927,155.547
C09843=1060.772,100.368,423.486,171.990,29.924,155.546
C09844=1060.766,100.119,423.504,171.988,29.922,155.546
C09845=1060.760,99.870,423.524,171.986,29.919,155.545
C09846=1060.754,99.621,423.542,171.985,29.917,155.545
C09847=1060.748,99.371,423.561,171.984,29.914,155.545
C09848=1060.741,99.122,423.580,171.982,29.912,155.544
C09849=1060.736,98.873,423.599,171.980,29.909,155.544
C09850=1060.729,98.624,423.618,171.979,29.906,155.544
C09851=1060.724,98.374,423.637,171.978,29.904,155.543
C09852=1060.717,98.125,423.656,171.976,29.901,155.543
C09853=1060.712,97.876,423.675,171.974,29.898,155.542
C09854=1060.706,97.627,423.693,171.973,29.896,155.542
C09855=1060.700,97.378,423.713,171.971,29.893,155.542
C09856=1060.694,97.129,423.731,171.969,29.891,155.541
C09857=1060.688,96.879,423.750,171.968,29.888,155.541
C09858=1060.682,96.630,423.769,171.967,29.885,155.540
C09859=1060.676,96.381,423.788,171.965,29.883,155.540
C09860=1060.669,96.131,423.807,171.963,29.880,155.540
C09861=1060.664,95.883,423.826,171.962,29.877,155.539
C09862=1060.658,95.634,423.845,171.961,29.875,155.539
C09863=1060.652,95.384,423.864,171.959,29.873,155.538
C09864=1060.646,95.135,423.882,171.957,29.870,155.538
C09865=1060.640,94.885,423.901,171.956,29.867,155.538
C09866=1060.633,94.601,423.922,171.954,29.864,155.537
C09867=1060.627,94.317,423.944,171.952,29.861,155.537
C09868=1060.620,94.032,423.965,171.951,29.858,155.536
C09869=1060.613,93.748,423.987,171.949,29.855,155.536
C09870=1060.607,93.499,424.005,171.947,29.852,155.535
C09871=1060.601,93.249,424.024,171.945,29.850,155.535
C09872=1060.595,93.000,424.043,171.944,29.847,155.535
C09873=1060.590,92.751,424.061,171.943,29.844,155.534
C09874=1060.584,92.502,424.080,171.941,29.842,155.534
C09875=1060.578,92.252,424.099,171.939,29.840,155.533
C09876=1060.571,92.003,424.118,171.938,29.837,155.533
C09877=1060.566,91.754,424.137,171.936,29.834,155.533
C09878=1060.560,91.505,424.155,171.935,29.832,155.532
C09879=1060.555,91.255,424.174,171.934,29.829,155.532
C09880=1060.548,91.006,424.193,171.932,29.826,155.531
C09881=1060.542,90.757,424.211,171.930,29.823,155.531
C09882=1060.537,90.508,424.229,171.928,29.821,155.531
C09883=1060.531,90.258,424.248,171.928,29.818,155.530
C09884=1060.524,90.009,424.267,171.926,29.816,155.530
C09885=1060.518,89.760,424.285,171.924,29.813,155.529
C09886=1060.512,89.510,424.304,171.923,29.811,155.529
C09887=1060.506,89.262,424.322,171.921,29.808,155.529
C09888=1060.500,89.013,424.341,171.920,29.805,155.528
C09889=1060.494,88.763,424.359,171.918,29.803,155.528
C09890=1060.488,88.513,424.378,171.917,29.800,155.528
C09891=1060.482,88.264,424.397,171.915,29.798,155.527
C09892=1060.476,88.015,424.414,171.913,29.795,155.527
C09893=1060.470,87.766,424.433,171.912,29.792,155.526
C09894=1060.463,87.517,424.451,171.911,29.790,155.526
C09895=1060.458,87.267,424.470,171.909,29.788,155.526
C09896=1060.452,87.019,424.488,171.907,29.785,155.525
C09897=1060.446,86.769,424.506,171.906,29.782,155.525
C09898=1060.440,86.520,424.525,171.905,29.780,155.524
C09899=1060.433,86.271,424.543,171.903,29.777,155.524
C09900=1060.428,86.021,424.562,171.901,29.774,155.524
C09901=1060.422,85.772,424.580,171.900,29.772,155.523
C09902=1060.416,85.522,424.598,171.898,29.769,155.523
C09903=1060.410,85.274,424.617,171.897,29.767,155.522
C09904=1060.404,85.024,424.634,171.895,29.764,155.522
C09905=1060.398,84.775,424.653,171.894,29.761,155.522
C09906=1060.392,84.526,424.672,171.892,29.759,155.521
C09907=1060.386,84.277,424.690,171.890,29.756,155.521
C09908=1060.380,84.027,424.709,171.890,29.754,155.521
C09909=1060.374,83.778,424.726,171.888,29.751,155.520
C09910=1060.368,83.529,424.745,171.886,29.748,155.520
C09911=1060.362,83.280,424.763,171.884,29.746,155.519
C09912=1060.356,83.030,424.782,171.884,29.743,155.519
C09913=1060.351,82.781,424.800,171.882,29.740,155.518
C09914=1060.344,82.532,424.818,171.880,29.738,155.518
C09915=1060.338,82.282,424.836,171.879,29.736,155.518
C09916=1060.333,82.033,424.854,171.877,29.733,155.517
C09917=1060.326,81.784,424.872,171.876,29.730,155.517
C09918=1060.321,81.534,424.891,171.874,29.728,155.517
C09919=1060.315,81.286,424.909,171.873,29.725,155.516
C09920=1060.309,81.036,424.927,171.871,29.722,155.516
C09921=1060.302,80.787,424.946,171.869,29.720,155.515
C09922=1060.297,80.538,424.963,171.869,29.717,155.515
C09923=1060.291,80.288,424.981,171.867,29.715,155.515
C09924=1060.285,80.040,424.999,171.865,29.712,155.514
C09925=1060.280,79.789,425.018,171.863,29.709,155.514
C09926=1060.273,79.540,425.037,171.863,29.707,155.513
C09927=1060.268,79.291,425.054,171.861,29.704,155.513
C09928=1060.262,79.042,425.072,171.859,29.701,155.513
C09929=1060.255,78.792,425.091,171.858,29.699,155.512
C09930=1060.248,78.508,425.111,171.856,29.696,155.512
C09931=1060.242,78.223,425.131,171.854,29.693,155.511
C09932=1060.235,77.939,425.152,171.853,29.690,155.511
C09933=1060.228,77.655,425.173,171.851,29.687,155.510
C09934=1060.222,77.405,425.191,171.849,29.684,155.510
C09935=1060.216,77.157,425.209,171.848,29.682,155.510
C09936=1060.210,76.907,425.227,171.847,29.680,155.509
C09937=1060.204,76.658,425.244,171.845,29.677,155.509
C09938=1060.198,76.408,425.262,171.843,29.674,155.509
C09939=1060.192,76.159,425.281,171.842,29.671,155.508
C09940=1060.186,75.910,425.298,171.841,29.669,155.508
C09941=1060.180,75.660,425.316,171.839,29.667,155.507
C09942=1060.173,75.411,425.334,171.837,29.664,155.507
C09943=1060.168,75.162,425.351,171.836,29.661,155.507
C09944=1060.162,74.913,425.370,171.834,29.658,155.506
C09945=1060.156,74.664,425.388,171.833,29.656,155.506
C09946=1060.150,74.414,425.406,171.831,29.654,155.506
C09947=1060.144,74.165,425.423,171.830,29.651,155.505
C09948=1060.138,73.915,425.441,171.828,29.648,155.505
C09949=1060.131,73.666,425.459,171.827,29.646,155.504
C09950=1060.126,73.417,425.477,171.826,29.644,155.504
C09951=1060.119,73.167,425.495,171.824,29.641,155.504
C09952=1060.114,72.918,425.512,171.822,29.638,155.503
C09953=1060.108,72.669,425.530,171.821,29.635,155.503
C09954=1060.102,72.420,425.548,171.820,29.633,155.502
C09955=1060.096,72.170,425.566,171.818,29.631,155.502
C09956=1060.090,71.921,425.584,171.816,29.628,155.502
C09957=1060.083,71.672,425.601,171.815,29.625,155.501
C09958=1060.078,71.423,425.619,171.814,29.623,155.501
C09959=1060.072,71.173,425.637,171.812,29.620,155.500
C09960=1060.066,70.924,425.654,171.810,29.618,155.500
C09961=1060.060,70.674,425.672,171.809,29.615,155.500
C09962=1060.054,70.425,425.690,171.807,29.612,155.499
C09963=1060.048,70.176,425.707,171.806,29.610,155.499
C09964=1060.042,69.926,425.725,171.805,29.607,155.499
C09965=1060.036,69.677,425.743,171.803,29.605,155.498
C09966=1060.030,69.427,425.761,171.801,29.602,155.498
C09967=1060.024,69.179,425.778,171.801,29.600,155.497
C09968=1060.018,68.929,425.795,171.799,29.597,155.497
C09969=1060.012,68.680,425.813,171.797,29.595,155.497
C09970=1060.006,68.430,425.831,171.795,29.592,155.496
C09971=1060.000,68.181,425.848,171.794,29.589,155.496
C09972=1059.994,67.932,425.866,171.793,29.587,155.496
C09973=1059.988,67.683,425.883,171.791,29.584,155.495
C09974=1059.981,67.433,425.901,171.790,29.582,155.495
C09975=1059.976,67.184,425.918,171.788,29.579,155.494
C09976=1059.970,66.934,425.936,171.787,29.576,155.494
C09977=1059.963,66.686,425.953,171.785,29.574,155.494
C09978=1059.957,66.436,425.971,171.784,29.571,155.493
C09979=1059.952,66.187,425.989,171.782,29.569,155.493
C09980=1059.945,65.938,426.006,171.781,29.566,155.493
C09981=1059.939,65.688,426.024,171.780,29.563,155.492
C09982=1059.934,65.439,426.041,171.778,29.561,155.492
C09983=1059.927,65.190,426.059,171.776,29.559,155.491
C09984=1059.922,64.940,426.075,171.774,29.556,155.491
C09985=1059.916,64.691,426.093,171.774,29.553,155.491
C09986=1059.909,64.442,426.110,171.772,29.551,155.490
C09987=1059.903,64.192,426.128,171.770,29.548,155.490
C09988=1059.897,63.943,426.145,171.769,29.546,155.490
C09989=1059.891,63.694,426.163,171.768,29.544,155.489
C09990=1059.885,63.445,426.180,171.766,29.541,155.489
C09991=1059.879,63.195,426.197,171.764,29.538,155.488
C09992=1059.873,62.946,426.214,171.763,29.536,155.488
C09993=1059.866,62.696,426.232,171.761,29.533,155.488
C09994=1059.859,62.412,426.252,171.759,29.530,155.487
C09995=1059.852,62.127,426.271,171.758,29.528,155.487
C09996=1059.845,61.842,426.291,171.756,29.525,155.487
//INST
///DATE 2021/06/25 14:46
///ATTR SC,RW,RJ
////FRAME ROBOT
///GROUP1 RB1
NOP
MOVL C00000 V=800.0 PL=0
MOVL C00001 V=800.0 PL=0
MOVL C00002 V=800.0 PL=0
MOVL C00003 V=800.0 PL=0
MOVL C00004 V=800.0 PL=0
MOVL C00005 V=800.0 PL=0
MOVL C00006 V=800.0 PL=0
MOVL C00007 V=800.0 PL=0
MOVL C00008 V=800.0 PL=0
MOVL C00009 V=800.0 PL=0
MOVL C00010 V=800.0 PL=0
MOVL C00011 V=800.0 PL=0
MOVL C00012 V=800.0 PL=0
MOVL C00013 V=800.0 PL=0
MOVL C00014 V=800.0 PL=0
MOVL C00015 V=800.0 PL=0
MOVL C00016 V=800.0 PL=0
MOVL C00017 V=800.0 PL=0
MOVL C00018 V=800.0 PL=0
MOVL C00019 V=800.0 PL=0
MOVL C00020 V=800.0 PL=0
MOVL C00021 V=800.0 PL=0
MOVL C00022 V=800.0 PL=0
MOVL C00023 V=800.0 PL=0
MOVL C00024 V=800.0 PL=0
MOVL C00025 V=800.0 PL=0
MOVL C00026 V=800.0 PL=0
MOVL C00027 V=800.0 PL=0
MOVL C00028 V=800.0 PL=0
MOVL C00029 V=800.0 PL=0
MOVL C00030 V=800.0 PL=0
MOVL C00031 V=800.0 PL=0
MOVL C00032 V=800.0 PL=0
MOVL C00033 V=800.0 PL=0
MOVL C00034 V=800.0 PL=0
MOVL C00035 V=800.0 PL=0
MOVL C00036 V=800.0 PL=0
MOVL C00037 V=800.0 PL=0
MOVL C00038 V=800.0 PL=0
MOVL C00039 V=800.0 PL=0
MOVL C00040 V=800.0 PL=0
MOVL C00041 V=800.0 PL=0
MOVL C00042 V=800.0 PL=0
MOVL C00043 V=800.0 PL=0
MOVL C00044 V=800.0 PL=0
MOVL C00045 V=800.0 PL=0
MOVL C00046 V=800.0 PL=0
MOVL C00047 V=800.0 PL=0
MOVL C00048 V=800.0 PL=0
MOVL C00049 V=800.0 PL=0
MOVL C00050 V=800.0 PL=0
MOVL C00051 V=800.0 PL=0
MOVL C00052 V=800.0 PL=0
MOVL C00053 V=800.0 PL=0
MOVL C00054 V=800.0 PL=0
MOVL C00055 V=800.0 PL=0
MOVL C00056 V=800.0 PL=0
MOVL C00057 V=800.0 PL=0
MOVL C00058 V=800.0 PL=0
MOVL C00059 V=800.0 PL=0
MOVL C00060 V=800.0 PL=0
MOVL C00061 V=800.0 PL=0
MOVL C00062 V=800.0 PL=0
MOVL C00063 V=800.0 PL=0
MOVL C00064 V=800.0 PL=0
MOVL C00065 V=800.0 PL=0
MOVL C00066 V=800.0 PL=0
MOVL C00067 V=800.0 PL=0
MOVL C00068 V=800.0 PL=0
MOVL C00069 V=800.0 PL=0
MOVL C00070 V=800.0 PL=0
MOVL C00071 V=800.0 PL=0
MOVL C00072 V=800.0 PL=0
MOVL C00073 V=800.0 PL=0
MOVL C00074 V=800.0 PL=0
MOVL C00075 V=800.0 PL=0
MOVL C00076 V=800.0 PL=0
MOVL C00077 V=800.0 PL=0
MOVL C00078 V=800.0 PL=0
MOVL C00079 V=800.0 PL=0
MOVL C00080 V=800.0 PL=0
MOVL C00081 V=800.0 PL=0
MOVL C00082 V=800.0 PL=0
MOVL C00083 V=800.0 PL=0
MOVL C00084 V=800.0 PL=0
MOVL C00085 V=800.0 PL=0
MOVL C00086 V=800.0 PL=0
MOVL C00087 V=800.0 PL=0
MOVL C00088 V=800.0 PL=0
MOVL C00089 V=800.0 PL=0
MOVL C00090 V=800.0 PL=0
MOVL C00091 V=800.0 PL=0
MOVL C00092 V=800.0 PL=0
MOVL C00093 V=800.0 PL=0
MOVL C00094 V=800.0 PL=0
MOVL C00095 V=800.0 PL=0
MOVL C00096 V=800.0 PL=0
MOVL C00097 V=800.0 PL=0
MOVL C00098 V=800.0 PL=0
MOVL C00099 V=800.0 PL=0
MOVL C00100 V=800.0 PL=0
MOVL C00101 V=800.0 PL=0
MOVL C00102 V=800.0 PL=0
MOVL C00103 V=800.0 PL=0
MOVL C00104 V=800.0 PL=0
MOVL C00105 V=800.0 PL=0
MOVL C00106 V=800.0 PL=0
MOVL C00107 V=800.0 PL=0
MOVL C00108 V=800.0 PL=0
MOVL C00109 V=800.0 PL=0
MOVL C00110 V=800.0 PL=0
MOVL C00111 V=800.0 PL=0
MOVL C00112 V=800.0 PL=0
MOVL C00113 V=800.0 PL=0
MOVL C00114 V=800.0 PL=0
MOVL C00115 V=800.0 PL=0
MOVL C00116 V=800.0 PL=0
MOVL C00117 V=800.0 PL=0
MOVL C00118 V=800.0 PL=0
MOVL C00119 V=800.0 PL=0
MOVL C00120 V=800.0 PL=0
MOVL C00121 V=800.0 PL=0
MOVL C00122 V=800.0 PL=0
MOVL C00123 V=800.0 PL=0
MOVL C00124 V=800.0 PL=0
MOVL C00125 V=800.0 PL=0
MOVL C00126 V=800.0 PL=0
MOVL C00127 V=800.0 PL=0
MOVL C00128 V=800.0 PL=0
MOVL C00129 V=800.0 PL=0
MOVL C00130 V=800.0 PL=0
MOVL C00131 V=800.0 PL=0
MOVL C00132 V=800.0 PL=0
MOVL C00133 V=800.0 PL=0
MOVL C00134 V=800.0 PL=0
MOVL C00135 V=800.0 PL=0
MOVL C00136 V=800.0 PL=0
MOVL C00137 V=800.0 PL=0
MOVL C00138 V=800.0 PL=0
MOVL C00139 V=800.0 PL=0
MOVL C00140 V=800.0 PL=0
MOVL C00141 V=800.0 PL=0
MOVL C00142 V=800.0 PL=0
MOVL C00143 V=800.0 PL=0
MOVL C00144 V=800.0 PL=0
MOVL C00145 V=800.0 PL=0
MOVL C00146 V=800.0 PL=0
MOVL C00147 V=800.0 PL=0
MOVL C00148 V=800.0 PL=0
MOVL C00149 V=800.0 PL=0
MOVL C00150 V=800.0 PL=0
MOVL C00151 V=800.0 PL=0
MOVL C00152 V=800.0 PL=0
MOVL C00153 V=800.0 PL=0
MOVL C00154 V=800.0 PL=0
MOVL C00155 V=800.0 PL=0
MOVL C00156 V=800.0 PL=0
MOVL C00157 V=800.0 PL=0
MOVL C00158 V=800.0 PL=0
MOVL C00159 V=800.0 PL=0
MOVL C00160 V=800.0 PL=0
MOVL C00161 V=800.0 PL=0
MOVL C00162 V=800.0 PL=0
MOVL C00163 V=800.0 PL=0
MOVL C00164 V=800.0 PL=0
MOVL C00165 V=800.0 PL=0
MOVL C00166 V=800.0 PL=0
MOVL C00167 V=800.0 PL=0
MOVL C00168 V=800.0 PL=0
MOVL C00169 V=800.0 PL=0
MOVL C00170 V=800.0 PL=0
MOVL C00171 V=800.0 PL=0
MOVL C00172 V=800.0 PL=0
MOVL C00173 V=800.0 PL=0
MOVL C00174 V=800.0 PL=0
MOVL C00175 V=800.0 PL=0
MOVL C00176 V=800.0 PL=0
MOVL C00177 V=800.0 PL=0
MOVL C00178 V=800.0 PL=0
MOVL C00179 V=800.0 PL=0
MOVL C00180 V=800.0 PL=0
MOVL C00181 V=800.0 PL=0
MOVL C00182 V=800.0 PL=0
MOVL C00183 V=800.0 PL=0
MOVL C00184 V=800.0 PL=0
MOVL C00185 V=800.0 PL=0
MOVL C00186 V=800.0 PL=0
MOVL C00187 V=800.0 PL=0
MOVL C00188 V=800.0 PL=0
MOVL C00189 V=800.0 PL=0
MOVL C00190 V=800.0 PL=0
MOVL C00191 V=800.0 PL=0
MOVL C00192 V=800.0 PL=0
MOVL C00193 V=800.0 PL=0
MOVL C00194 V=800.0 PL=0
MOVL C00195 V=800.0 PL=0
MOVL C00196 V=800.0 PL=0
MOVL C00197 V=800.0 PL=0
MOVL C00198 V=800.0 PL=0
MOVL C00199 V=800.0 PL=0
MOVL C00200 V=800.0 PL=0
MOVL C00201 V=800.0 PL=0
MOVL C00202 V=800.0 PL=0
MOVL C00203 V=800.0 PL=0
MOVL C00204 V=800.0 PL=0
MOVL C00205 V=800.0 PL=0
MOVL C00206 V=800.0 PL=0
MOVL C00207 V=800.0 PL=0
MOVL C00208 V=800.0 PL=0
MOVL C00209 V=800.0 PL=0
MOVL C00210 V=800.0 PL=0
MOVL C00211 V=800.0 PL=0
MOVL C00212 V=800.0 PL=0
MOVL C00213 V=800.0 PL=0
MOVL C00214 V=800.0 PL=0
MOVL C00215 V=800.0 PL=0
MOVL C00216 V=800.0 PL=0
MOVL C00217 V=800.0 PL=0
MOVL C00218 V=800.0 PL=0
MOVL C00219 V=800.0 PL=0
MOVL C00220 V=800.0 PL=0
MOVL C00221 V=800.0 PL=0
MOVL C00222 V=800.0 PL=0
MOVL C00223 V=800.0 PL=0
MOVL C00224 V=800.0 PL=0
MOVL C00225 V=800.0 PL=0
MOVL C00226 V=800.0 PL=0
MOVL C00227 V=800.0 PL=0
MOVL C00228 V=800.0 PL=0
MOVL C00229 V=800.0 PL=0
MOVL C00230 V=800.0 PL=0
MOVL C00231 V=800.0 PL=0
MOVL C00232 V=800.0 PL=0
MOVL C00233 V=800.0 PL=0
MOVL C00234 V=800.0 PL=0
MOVL C00235 V=800.0 PL=0
MOVL C00236 V=800.0 PL=0
MOVL C00237 V=800.0 PL=0
MOVL C00238 V=800.0 PL=0
MOVL C00239 V=800.0 PL=0
MOVL C00240 V=800.0 PL=0
MOVL C00241 V=800.0 PL=0
MOVL C00242 V=800.0 PL=0
MOVL C00243 V=800.0 PL=0
MOVL C00244 V=800.0 PL=0
MOVL C00245 V=800.0 PL=0
MOVL C00246 V=800.0 PL=0
MOVL C00247 V=800.0 PL=0
MOVL C00248 V=800.0 PL=0
MOVL C00249 V=800.0 PL=0
MOVL C00250 V=800.0 PL=0
MOVL C00251 V=800.0 PL=0
MOVL C00252 V=800.0 PL=0
MOVL C00253 V=800.0 PL=0
MOVL C00254 V=800.0 PL=0
MOVL C00255 V=800.0 PL=0
MOVL C00256 V=800.0 PL=0
MOVL C00257 V=800.0 PL=0
MOVL C00258 V=800.0 PL=0
MOVL C00259 V=800.0 PL=0
MOVL C00260 V=800.0 PL=0
MOVL C00261 V=800.0 PL=0
MOVL C00262 V=800.0 PL=0
MOVL C00263 V=800.0 PL=0
MOVL C00264 V=800.0 PL=0
MOVL C00265 V=800.0 PL=0
MOVL C00266 V=800.0 PL=0
MOVL C00267 V=800.0 PL=0
MOVL C00268 V=800.0 PL=0
MOVL C00269 V=800.0 PL=0
MOVL C00270 V=800.0 PL=0
MOVL C00271 V=800.0 PL=0
MOVL C00272 V=800.0 PL=0
MOVL C00273 V=800.0 PL=0
MOVL C00274 V=800.0 PL=0
MOVL C00275 V=800.0 PL=0
MOVL C00276 V=800.0 PL=0
MOVL C00277 V=800.0 PL=0
MOVL C00278 V=800.0 PL=0
MOVL C00279 V=800.0 PL=0
MOVL C00280 V=800.0 PL=0
MOVL C00281 V=800.0 PL=0
MOVL C00282 V=800.0 PL=0
MOVL C00283 V=800.0 PL=0
MOVL C00284 V=800.0 PL=0
MOVL C00285 V=800.0 PL=0
MOVL C00286 V=800.0 PL=0
MOVL C00287 V=800.0 PL=0
MOVL C00288 V=800.0 PL=0
MOVL C00289 V=800.0 PL=0
MOVL C00290 V=800.0 PL=0
MOVL C00291 V=800.0 PL=0
MOVL C00292 V=800.0 PL=0
MOVL C00293 V=800.0 PL=0
MOVL C00294 V=800.0 PL=0
MOVL C00295 V=800.0 PL=0
MOVL C00296 V=800.0 PL=0
MOVL C00297 V=800.0 PL=0
MOVL C00298 V=800.0 PL=0
MOVL C00299 V=800.0 PL=0
MOVL C00300 V=800.0 PL=0
MOVL C00301 V=800.0 PL=0
MOVL C00302 V=800.0 PL=0
MOVL C00303 V=800.0 PL=0
MOVL C00304 V=800.0 PL=0
MOVL C00305 V=800.0 PL=0
MOVL C00306 V=800.0 PL=0
MOVL C00307 V=800.0 PL=0
MOVL C00308 V=800.0 PL=0
MOVL C00309 V=800.0 PL=0
MOVL C00310 V=800.0 PL=0
MOVL C00311 V=800.0 PL=0
MOVL C00312 V=800.0 PL=0
MOVL C00313 V=800.0 PL=0
MOVL C00314 V=800.0 PL=0
MOVL C00315 V=800.0 PL=0
MOVL C00316 V=800.0 PL=0
MOVL C00317 V=800.0 PL=0
MOVL C00318 V=800.0 PL=0
MOVL C00319 V=800.0 PL=0
MOVL C00320 V=800.0 PL=0
MOVL C00321 V=800.0 PL=0
MOVL C00322 V=800.0 PL=0
MOVL C00323 V=800.0 PL=0
MOVL C00324 V=800.0 PL=0
MOVL C00325 V=800.0 PL=0
MOVL C00326 V=800.0 PL=0
MOVL C00327 V=800.0 PL=0
MOVL C00328 V=800.0 PL=0
MOVL C00329 V=800.0 PL=0
MOVL C00330 V=800.0 PL=0
MOVL C00331 V=800.0 PL=0
MOVL C00332 V=800.0 PL=0
MOVL C00333 V=800.0 PL=0
MOVL C00334 V=800.0 PL=0
MOVL C00335 V=800.0 PL=0
MOVL C00336 V=800.0 PL=0
MOVL C00337 V=800.0 PL=0
MOVL C00338 V=800.0 PL=0
MOVL C00339 V=800.0 PL=0
MOVL C00340 V=800.0 PL=0
MOVL C00341 V=800.0 PL=0
MOVL C00342 V=800.0 PL=0
MOVL C00343 V=800.0 PL=0
MOVL C00344 V=800.0 PL=0
MOVL C00345 V=800.0 PL=0
MOVL C00346 V=800.0 PL=0
MOVL C00347 V=800.0 PL=0
MOVL C00348 V=800.0 PL=0
MOVL C00349 V=800.0 PL=0
MOVL C00350 V=800.0 PL=0
MOVL C00351 V=800.0 PL=0
MOVL C00352 V=800.0 PL=0
MOVL C00353 V=800.0 PL=0
MOVL C00354 V=800.0 PL=0
MOVL C00355 V=800.0 PL=0
MOVL C00356 V=800.0 PL=0
MOVL C00357 V=800.0 PL=0
MOVL C00358 V=800.0 PL=0
MOVL C00359 V=800.0 PL=0
MOVL C00360 V=800.0 PL=0
MOVL C00361 V=800.0 PL=0
MOVL C00362 V=800.0 PL=0
MOVL C00363 V=800.0 PL=0
MOVL C00364 V=800.0 PL=0
MOVL C00365 V=800.0 PL=0
MOVL C00366 V=800.0 PL=0
MOVL C00367 V=800.0 PL=0
MOVL C00368 V=800.0 PL=0
MOVL C00369 V=800.0 PL=0
MOVL C00370 V=800.0 PL=0
MOVL C00371 V=800.0 PL=0
MOVL C00372 V=800.0 PL=0
MOVL C00373 V=800.0 PL=0
MOVL C00374 V=800.0 PL=0
MOVL C00375 V=800.0 PL=0
MOVL C00376 V=800.0 PL=0
MOVL C00377 V=800.0 PL=0
MOVL C00378 V=800.0 PL=0
MOVL C00379 V=800.0 PL=0
MOVL C00380 V=800.0 PL=0
MOVL C00381 V=800.0 PL=0
MOVL C00382 V=800.0 PL=0
MOVL C00383 V=800.0 PL=0
MOVL C00384 V=800.0 PL=0
MOVL C00385 V=800.0 PL=0
MOVL C00386 V=800.0 PL=0
MOVL C00387 V=800.0 PL=0
MOVL C00388 V=800.0 PL=0
MOVL C00389 V=800.0 PL=0
MOVL C00390 V=800.0 PL=0
MOVL C00391 V=800.0 PL=0
MOVL C00392 V=800.0 PL=0
MOVL C00393 V=800.0 PL=0
MOVL C00394 V=800.0 PL=0
MOVL C00395 V=800.0 PL=0
MOVL C00396 V=800.0 PL=0
MOVL C00397 V=800.0 PL=0
MOVL C00398 V=800.0 PL=0
MOVL C00399 V=800.0 PL=0
MOVL C00400 V=800.0 PL=0
MOVL C00401 V=800.0 PL=0
MOVL C00402 V=800.0 PL=0
MOVL C00403 V=800.0 PL=0
MOVL C00404 V=800.0 PL=0
MOVL C00405 V=800.0 PL=0
MOVL C00406 V=800.0 PL=0
MOVL C00407 V=800.0 PL=0
MOVL C00408 V=800.0 PL=0
MOVL C00409 V=800.0 PL=0
MOVL C00410 V=800.0 PL=0
MOVL C00411 V=800.0 PL=0
MOVL C00412 V=800.0 PL=0
MOVL C00413 V=800.0 PL=0
MOVL C00414 V=800.0 PL=0
MOVL C00415 V=800.0 PL=0
MOVL C00416 V=800.0 PL=0
MOVL C00417 V=800.0 PL=0
MOVL C00418 V=800.0 PL=0
MOVL C00419 V=800.0 PL=0
MOVL C00420 V=800.0 PL=0
MOVL C00421 V=800.0 PL=0
MOVL C00422 V=800.0 PL=0
MOVL C00423 V=800.0 PL=0
MOVL C00424 V=800.0 PL=0
MOVL C00425 V=800.0 PL=0
MOVL C00426 V=800.0 PL=0
MOVL C00427 V=800.0 PL=0
MOVL C00428 V=800.0 PL=0
MOVL C00429 V=800.0 PL=0
MOVL C00430 V=800.0 PL=0
MOVL C00431 V=800.0 PL=0
MOVL C00432 V=800.0 PL=0
MOVL C00433 V=800.0 PL=0
MOVL C00434 V=800.0 PL=0
MOVL C00435 V=800.0 PL=0
MOVL C00436 V=800.0 PL=0
MOVL C00437 V=800.0 PL=0
MOVL C00438 V=800.0 PL=0
MOVL C00439 V=800.0 PL=0
MOVL C00440 V=800.0 PL=0
MOVL C00441 V=800.0 PL=0
MOVL C00442 V=800.0 PL=0
MOVL C00443 V=800.0 PL=0
MOVL C00444 V=800.0 PL=0
MOVL C00445 V=800.0 PL=0
MOVL C00446 V=800.0 PL=0
MOVL C00447 V=800.0 PL=0
MOVL C00448 V=800.0 PL=0
MOVL C00449 V=800.0 PL=0
MOVL C00450 V=800.0 PL=0
MOVL C00451 V=800.0 PL=0
MOVL C00452 V=800.0 PL=0
MOVL C00453 V=800.0 PL=0
MOVL C00454 V=800.0 PL=0
MOVL C00455 V=800.0 PL=0
MOVL C00456 V=800.0 PL=0
MOVL C00457 V=800.0 PL=0
MOVL C00458 V=800.0 PL=0
MOVL C00459 V=800.0 PL=0
MOVL C00460 V=800.0 PL=0
MOVL C00461 V=800.0 PL=0
MOVL C00462 V=800.0 PL=0
MOVL C00463 V=800.0 PL=0
MOVL C00464 V=800.0 PL=0
MOVL C00465 V=800.0 PL=0
MOVL C00466 V=800.0 PL=0
MOVL C00467 V=800.0 PL=0
MOVL C00468 V=800.0 PL=0
MOVL C00469 V=800.0 PL=0
MOVL C00470 V=800.0 PL=0
MOVL C00471 V=800.0 PL=0
MOVL C00472 V=800.0 PL=0
MOVL C00473 V=800.0 PL=0
MOVL C00474 V=800.0 PL=0
MOVL C00475 V=800.0 PL=0
MOVL C00476 V=800.0 PL=0
MOVL C00477 V=800.0 PL=0
MOVL C00478 V=800.0 PL=0
MOVL C00479 V=800.0 PL=0
MOVL C00480 V=800.0 PL=0
MOVL C00481 V=800.0 PL=0
MOVL C00482 V=800.0 PL=0
MOVL C00483 V=800.0 PL=0
MOVL C00484 V=800.0 PL=0
MOVL C00485 V=800.0 PL=0
MOVL C00486 V=800.0 PL=0
MOVL C00487 V=800.0 PL=0
MOVL C00488 V=800.0 PL=0
MOVL C00489 V=800.0 PL=0
MOVL C00490 V=800.0 PL=0
MOVL C00491 V=800.0 PL=0
MOVL C00492 V=800.0 PL=0
MOVL C00493 V=800.0 PL=0
MOVL C00494 V=800.0 PL=0
MOVL C00495 V=800.0 PL=0
MOVL C00496 V=800.0 PL=0
MOVL C00497 V=800.0 PL=0
MOVL C00498 V=800.0 PL=0
MOVL C00499 V=800.0 PL=0
MOVL C00500 V=800.0 PL=0
MOVL C00501 V=800.0 PL=0
MOVL C00502 V=800.0 PL=0
MOVL C00503 V=800.0 PL=0
MOVL C00504 V=800.0 PL=0
MOVL C00505 V=800.0 PL=0
MOVL C00506 V=800.0 PL=0
MOVL C00507 V=800.0 PL=0
MOVL C00508 V=800.0 PL=0
MOVL C00509 V=800.0 PL=0
MOVL C00510 V=800.0 PL=0
MOVL C00511 V=800.0 PL=0
MOVL C00512 V=800.0 PL=0
MOVL C00513 V=800.0 PL=0
MOVL C00514 V=800.0 PL=0
MOVL C00515 V=800.0 PL=0
MOVL C00516 V=800.0 PL=0
MOVL C00517 V=800.0 PL=0
MOVL C00518 V=800.0 PL=0
MOVL C00519 V=800.0 PL=0
MOVL C00520 V=800.0 PL=0
MOVL C00521 V=800.0 PL=0
MOVL C00522 V=800.0 PL=0
MOVL C00523 V=800.0 PL=0
MOVL C00524 V=800.0 PL=0
MOVL C00525 V=800.0 PL=0
MOVL C00526 V=800.0 PL=0
MOVL C00527 V=800.0 PL=0
MOVL C00528 V=800.0 PL=0
MOVL C00529 V=800.0 PL=0
MOVL C00530 V=800.0 PL=0
MOVL C00531 V=800.0 PL=0
MOVL C00532 V=800.0 PL=0
MOVL C00533 V=800.0 PL=0
MOVL C00534 V=800.0 PL=0
MOVL C00535 V=800.0 PL=0
MOVL C00536 V=800.0 PL=0
MOVL C00537 V=800.0 PL=0
MOVL C00538 V=800.0 PL=0
MOVL C00539 V=800.0 PL=0
MOVL C00540 V=800.0 PL=0
MOVL C00541 V=800.0 PL=0
MOVL C00542 V=800.0 PL=0
MOVL C00543 V=800.0 PL=0
MOVL C00544 V=800.0 PL=0
MOVL C00545 V=800.0 PL=0
MOVL C00546 V=800.0 PL=0
MOVL C00547 V=800.0 PL=0
MOVL C00548 V=800.0 PL=0
MOVL C00549 V=800.0 PL=0
MOVL C00550 V=800.0 PL=0
MOVL C00551 V=800.0 PL=0
MOVL C00552 V=800.0 PL=0
MOVL C00553 V=800.0 PL=0
MOVL C00554 V=800.0 PL=0
MOVL C00555 V=800.0 PL=0
MOVL C00556 V=800.0 PL=0
MOVL C00557 V=800.0 PL=0
MOVL C00558 V=800.0 PL=0
MOVL C00559 V=800.0 PL=0
MOVL C00560 V=800.0 PL=0
MOVL C00561 V=800.0 PL=0
MOVL C00562 V=800.0 PL=0
MOVL C00563 V=800.0 PL=0
MOVL C00564 V=800.0 PL=0
MOVL C00565 V=800.0 PL=0
MOVL C00566 V=800.0 PL=0
MOVL C00567 V=800.0 PL=0
MOVL C00568 V=800.0 PL=0
MOVL C00569 V=800.0 PL=0
MOVL C00570 V=800.0 PL=0
MOVL C00571 V=800.0 PL=0
MOVL C00572 V=800.0 PL=0
MOVL C00573 V=800.0 PL=0
MOVL C00574 V=800.0 PL=0
MOVL C00575 V=800.0 PL=0
MOVL C00576 V=800.0 PL=0
MOVL C00577 V=800.0 PL=0
MOVL C00578 V=800.0 PL=0
MOVL C00579 V=800.0 PL=0
MOVL C00580 V=800.0 PL=0
MOVL C00581 V=800.0 PL=0
MOVL C00582 V=800.0 PL=0
MOVL C00583 V=800.0 PL=0
MOVL C00584 V=800.0 PL=0
MOVL C00585 V=800.0 PL=0
MOVL C00586 V=800.0 PL=0
MOVL C00587 V=800.0 PL=0
MOVL C00588 V=800.0 PL=0
MOVL C00589 V=800.0 PL=0
MOVL C00590 V=800.0 PL=0
MOVL C00591 V=800.0 PL=0
MOVL C00592 V=800.0 PL=0
MOVL C00593 V=800.0 PL=0
MOVL C00594 V=800.0 PL=0
MOVL C00595 V=800.0 PL=0
MOVL C00596 V=800.0 PL=0
MOVL C00597 V=800.0 PL=0
MOVL C00598 V=800.0 PL=0
MOVL C00599 V=800.0 PL=0
MOVL C00600 V=800.0 PL=0
MOVL C00601 V=800.0 PL=0
MOVL C00602 V=800.0 PL=0
MOVL C00603 V=800.0 PL=0
MOVL C00604 V=800.0 PL=0
MOVL C00605 V=800.0 PL=0
MOVL C00606 V=800.0 PL=0
MOVL C00607 V=800.0 PL=0
MOVL C00608 V=800.0 PL=0
MOVL C00609 V=800.0 PL=0
MOVL C00610 V=800.0 PL=0
MOVL C00611 V=800.0 PL=0
MOVL C00612 V=800.0 PL=0
MOVL C00613 V=800.0 PL=0
MOVL C00614 V=800.0 PL=0
MOVL C00615 V=800.0 PL=0
MOVL C00616 V=800.0 PL=0
MOVL C00617 V=800.0 PL=0
MOVL C00618 V=800.0 PL=0
MOVL C00619 V=800.0 PL=0
MOVL C00620 V=800.0 PL=0
MOVL C00621 V=800.0 PL=0
MOVL C00622 V=800.0 PL=0
MOVL C00623 V=800.0 PL=0
MOVL C00624 V=800.0 PL=0
MOVL C00625 V=800.0 PL=0
MOVL C00626 V=800.0 PL=0
MOVL C00627 V=800.0 PL=0
MOVL C00628 V=800.0 PL=0
MOVL C00629 V=800.0 PL=0
MOVL C00630 V=800.0 PL=0
MOVL C00631 V=800.0 PL=0
MOVL C00632 V=800.0 PL=0
MOVL C00633 V=800.0 PL=0
MOVL C00634 V=800.0 PL=0
MOVL C00635 V=800.0 PL=0
MOVL C00636 V=800.0 PL=0
MOVL C00637 V=800.0 PL=0
MOVL C00638 V=800.0 PL=0
MOVL C00639 V=800.0 PL=0
MOVL C00640 V=800.0 PL=0
MOVL C00641 V=800.0 PL=0
MOVL C00642 V=800.0 PL=0
MOVL C00643 V=800.0 PL=0
MOVL C00644 V=800.0 PL=0
MOVL C00645 V=800.0 PL=0
MOVL C00646 V=800.0 PL=0
MOVL C00647 V=800.0 PL=0
MOVL C00648 V=800.0 PL=0
MOVL C00649 V=800.0 PL=0
MOVL C00650 V=800.0 PL=0
MOVL C00651 V=800.0 PL=0
MOVL C00652 V=800.0 PL=0
MOVL C00653 V=800.0 PL=0
MOVL C00654 V=800.0 PL=0
MOVL C00655 V=800.0 PL=0
MOVL C00656 V=800.0 PL=0
MOVL C00657 V=800.0 PL=0
MOVL C00658 V=800.0 PL=0
MOVL C00659 V=800.0 PL=0
MOVL C00660 V=800.0 PL=0
MOVL C00661 V=800.0 PL=0
MOVL C00662 V=800.0 PL=0
MOVL C00663 V=800.0 PL=0
MOVL C00664 V=800.0 PL=0
MOVL C00665 V=800.0 PL=0
MOVL C00666 V=800.0 PL=0
MOVL C00667 V=800.0 PL=0
MOVL C00668 V=800.0 PL=0
MOVL C00669 V=800.0 PL=0
MOVL C00670 V=800.0 PL=0
MOVL C00671 V=800.0 PL=0
MOVL C00672 V=800.0 PL=0
MOVL C00673 V=800.0 PL=0
MOVL C00674 V=800.0 PL=0
MOVL C00675 V=800.0 PL=0
MOVL C00676 V=800.0 PL=0
MOVL C00677 V=800.0 PL=0
MOVL C00678 V=800.0 PL=0
MOVL C00679 V=800.0 PL=0
MOVL C00680 V=800.0 PL=0
MOVL C00681 V=800.0 PL=0
MOVL C00682 V=800.0 PL=0
MOVL C00683 V=800.0 PL=0
MOVL C00684 V=800.0 PL=0
MOVL C00685 V=800.0 PL=0
MOVL C00686 V=800.0 PL=0
MOVL C00687 V=800.0 PL=0
MOVL C00688 V=800.0 PL=0
MOVL C00689 V=800.0 PL=0
MOVL C00690 V=800.0 PL=0
MOVL C00691 V=800.0 PL=0
MOVL C00692 V=800.0 PL=0
MOVL C00693 V=800.0 PL=0
MOVL C00694 V=800.0 PL=0
MOVL C00695 V=800.0 PL=0
MOVL C00696 V=800.0 PL=0
MOVL C00697 V=800.0 PL=0
MOVL C00698 V=800.0 PL=0
MOVL C00699 V=800.0 PL=0
MOVL C00700 V=800.0 PL=0
MOVL C00701 V=800.0 PL=0
MOVL C00702 V=800.0 PL=0
MOVL C00703 V=800.0 PL=0
MOVL C00704 V=800.0 PL=0
MOVL C00705 V=800.0 PL=0
MOVL C00706 V=800.0 PL=0
MOVL C00707 V=800.0 PL=0
MOVL C00708 V=800.0 PL=0
MOVL C00709 V=800.0 PL=0
MOVL C00710 V=800.0 PL=0
MOVL C00711 V=800.0 PL=0
MOVL C00712 V=800.0 PL=0
MOVL C00713 V=800.0 PL=0
MOVL C00714 V=800.0 PL=0
MOVL C00715 V=800.0 PL=0
MOVL C00716 V=800.0 PL=0
MOVL C00717 V=800.0 PL=0
MOVL C00718 V=800.0 PL=0
MOVL C00719 V=800.0 PL=0
MOVL C00720 V=800.0 PL=0
MOVL C00721 V=800.0 PL=0
MOVL C00722 V=800.0 PL=0
MOVL C00723 V=800.0 PL=0
MOVL C00724 V=800.0 PL=0
MOVL C00725 V=800.0 PL=0
MOVL C00726 V=800.0 PL=0
MOVL C00727 V=800.0 PL=0
MOVL C00728 V=800.0 PL=0
MOVL C00729 V=800.0 PL=0
MOVL C00730 V=800.0 PL=0
MOVL C00731 V=800.0 PL=0
MOVL C00732 V=800.0 PL=0
MOVL C00733 V=800.0 PL=0
MOVL C00734 V=800.0 PL=0
MOVL C00735 V=800.0 PL=0
MOVL C00736 V=800.0 PL=0
MOVL C00737 V=800.0 PL=0
MOVL C00738 V=800.0 PL=0
MOVL C00739 V=800.0 PL=0
MOVL C00740 V=800.0 PL=0
MOVL C00741 V=800.0 PL=0
MOVL C00742 V=800.0 PL=0
MOVL C00743 V=800.0 PL=0
MOVL C00744 V=800.0 PL=0
MOVL C00745 V=800.0 PL=0
MOVL C00746 V=800.0 PL=0
MOVL C00747 V=800.0 PL=0
MOVL C00748 V=800.0 PL=0
MOVL C00749 V=800.0 PL=0
MOVL C00750 V=800.0 PL=0
MOVL C00751 V=800.0 PL=0
MOVL C00752 V=800.0 PL=0
MOVL C00753 V=800.0 PL=0
MOVL C00754 V=800.0 PL=0
MOVL C00755 V=800.0 PL=0
MOVL C00756 V=800.0 PL=0
MOVL C00757 V=800.0 PL=0
MOVL C00758 V=800.0 PL=0
MOVL C00759 V=800.0 PL=0
MOVL C00760 V=800.0 PL=0
MOVL C00761 V=800.0 PL=0
MOVL C00762 V=800.0 PL=0
MOVL C00763 V=800.0 PL=0
MOVL C00764 V=800.0 PL=0
MOVL C00765 V=800.0 PL=0
MOVL C00766 V=800.0 PL=0
MOVL C00767 V=800.0 PL=0
MOVL C00768 V=800.0 PL=0
MOVL C00769 V=800.0 PL=0
MOVL C00770 V=800.0 PL=0
MOVL C00771 V=800.0 PL=0
MOVL C00772 V=800.0 PL=0
MOVL C00773 V=800.0 PL=0
MOVL C00774 V=800.0 PL=0
MOVL C00775 V=800.0 PL=0
MOVL C00776 V=800.0 PL=0
MOVL C00777 V=800.0 PL=0
MOVL C00778 V=800.0 PL=0
MOVL C00779 V=800.0 PL=0
MOVL C00780 V=800.0 PL=0
MOVL C00781 V=800.0 PL=0
MOVL C00782 V=800.0 PL=0
MOVL C00783 V=800.0 PL=0
MOVL C00784 V=800.0 PL=0
MOVL C00785 V=800.0 PL=0
MOVL C00786 V=800.0 PL=0
MOVL C00787 V=800.0 PL=0
MOVL C00788 V=800.0 PL=0
MOVL C00789 V=800.0 PL=0
MOVL C00790 V=800.0 PL=0
MOVL C00791 V=800.0 PL=0
MOVL C00792 V=800.0 PL=0
MOVL C00793 V=800.0 PL=0
MOVL C00794 V=800.0 PL=0
MOVL C00795 V=800.0 PL=0
MOVL C00796 V=800.0 PL=0
MOVL C00797 V=800.0 PL=0
MOVL C00798 V=800.0 PL=0
MOVL C00799 V=800.0 PL=0
MOVL C00800 V=800.0 PL=0
MOVL C00801 V=800.0 PL=0
MOVL C00802 V=800.0 PL=0
MOVL C00803 V=800.0 PL=0
MOVL C00804 V=800.0 PL=0
MOVL C00805 V=800.0 PL=0
MOVL C00806 V=800.0 PL=0
MOVL C00807 V=800.0 PL=0
MOVL C00808 V=800.0 PL=0
MOVL C00809 V=800.0 PL=0
MOVL C00810 V=800.0 PL=0
MOVL C00811 V=800.0 PL=0
MOVL C00812 V=800.0 PL=0
MOVL C00813 V=800.0 PL=0
MOVL C00814 V=800.0 PL=0
MOVL C00815 V=800.0 PL=0
MOVL C00816 V=800.0 PL=0
MOVL C00817 V=800.0 PL=0
MOVL C00818 V=800.0 PL=0
MOVL C00819 V=800.0 PL=0
MOVL C00820 V=800.0 PL=0
MOVL C00821 V=800.0 PL=0
MOVL C00822 V=800.0 PL=0
MOVL C00823 V=800.0 PL=0
MOVL C00824 V=800.0 PL=0
MOVL C00825 V=800.0 PL=0
MOVL C00826 V=800.0 PL=0
MOVL C00827 V=800.0 PL=0
MOVL C00828 V=800.0 PL=0
MOVL C00829 V=800.0 PL=0
MOVL C00830 V=800.0 PL=0
MOVL C00831 V=800.0 PL=0
MOVL C00832 V=800.0 PL=0
MOVL C00833 V=800.0 PL=0
MOVL C00834 V=800.0 PL=0
MOVL C00835 V=800.0 PL=0
MOVL C00836 V=800.0 PL=0
MOVL C00837 V=800.0 PL=0
MOVL C00838 V=800.0 PL=0
MOVL C00839 V=800.0 PL=0
MOVL C00840 V=800.0 PL=0
MOVL C00841 V=800.0 PL=0
MOVL C00842 V=800.0 PL=0
MOVL C00843 V=800.0 PL=0
MOVL C00844 V=800.0 PL=0
MOVL C00845 V=800.0 PL=0
MOVL C00846 V=800.0 PL=0
MOVL C00847 V=800.0 PL=0
MOVL C00848 V=800.0 PL=0
MOVL C00849 V=800.0 PL=0
MOVL C00850 V=800.0 PL=0
MOVL C00851 V=800.0 PL=0
MOVL C00852 V=800.0 PL=0
MOVL C00853 V=800.0 PL=0
MOVL C00854 V=800.0 PL=0
MOVL C00855 V=800.0 PL=0
MOVL C00856 V=800.0 PL=0
MOVL C00857 V=800.0 PL=0
MOVL C00858 V=800.0 PL=0
MOVL C00859 V=800.0 PL=0
MOVL C00860 V=800.0 PL=0
MOVL C00861 V=800.0 PL=0
MOVL C00862 V=800.0 PL=0
MOVL C00863 V=800.0 PL=0
MOVL C00864 V=800.0 PL=0
MOVL C00865 V=800.0 PL=0
MOVL C00866 V=800.0 PL=0
MOVL C00867 V=800.0 PL=0
MOVL C00868 V=800.0 PL=0
MOVL C00869 V=800.0 PL=0
MOVL C00870 V=800.0 PL=0
MOVL C00871 V=800.0 PL=0
MOVL C00872 V=800.0 PL=0
MOVL C00873 V=800.0 PL=0
MOVL C00874 V=800.0 PL=0
MOVL C00875 V=800.0 PL=0
MOVL C00876 V=800.0 PL=0
MOVL C00877 V=800.0 PL=0
MOVL C00878 V=800.0 PL=0
MOVL C00879 V=800.0 PL=0
MOVL C00880 V=800.0 PL=0
MOVL C00881 V=800.0 PL=0
MOVL C00882 V=800.0 PL=0
MOVL C00883 V=800.0 PL=0
MOVL C00884 V=800.0 PL=0
MOVL C00885 V=800.0 PL=0
MOVL C00886 V=800.0 PL=0
MOVL C00887 V=800.0 PL=0
MOVL C00888 V=800.0 PL=0
MOVL C00889 V=800.0 PL=0
MOVL C00890 V=800.0 PL=0
MOVL C00891 V=800.0 PL=0
MOVL C00892 V=800.0 PL=0
MOVL C00893 V=800.0 PL=0
MOVL C00894 V=800.0 PL=0
MOVL C00895 V=800.0 PL=0
MOVL C00896 V=800.0 PL=0
MOVL C00897 V=800.0 PL=0
MOVL C00898 V=800.0 PL=0
MOVL C00899 V=800.0 PL=0
MOVL C00900 V=800.0 PL=0
MOVL C00901 V=800.0 PL=0
MOVL C00902 V=800.0 PL=0
MOVL C00903 V=800.0 PL=0
MOVL C00904 V=800.0 PL=0
MOVL C00905 V=800.0 PL=0
MOVL C00906 V=800.0 PL=0
MOVL C00907 V=800.0 PL=0
MOVL C00908 V=800.0 PL=0
MOVL C00909 V=800.0 PL=0
MOVL C00910 V=800.0 PL=0
MOVL C00911 V=800.0 PL=0
MOVL C00912 V=800.0 PL=0
MOVL C00913 V=800.0 PL=0
MOVL C00914 V=800.0 PL=0
MOVL C00915 V=800.0 PL=0
MOVL C00916 V=800.0 PL=0
MOVL C00917 V=800.0 PL=0
MOVL C00918 V=800.0 PL=0
MOVL C00919 V=800.0 PL=0
MOVL C00920 V=800.0 PL=0
MOVL C00921 V=800.0 PL=0
MOVL C00922 V=800.0 PL=0
MOVL C00923 V=800.0 PL=0
MOVL C00924 V=800.0 PL=0
MOVL C00925 V=800.0 PL=0
MOVL C00926 V=800.0 PL=0
MOVL C00927 V=800.0 PL=0
MOVL C00928 V=800.0 PL=0
MOVL C00929 V=800.0 PL=0
MOVL C00930 V=800.0 PL=0
MOVL C00931 V=800.0 PL=0
MOVL C00932 V=800.0 PL=0
MOVL C00933 V=800.0 PL=0
MOVL C00934 V=800.0 PL=0
MOVL C00935 V=800.0 PL=0
MOVL C00936 V=800.0 PL=0
MOVL C00937 V=800.0 PL=0
MOVL C00938 V=800.0 PL=0
MOVL C00939 V=800.0 PL=0
MOVL C00940 V=800.0 PL=0
MOVL C00941 V=800.0 PL=0
MOVL C00942 V=800.0 PL=0
MOVL C00943 V=800.0 PL=0
MOVL C00944 V=800.0 PL=0
MOVL C00945 V=800.0 PL=0
MOVL C00946 V=800.0 PL=0
MOVL C00947 V=800.0 PL=0
MOVL C00948 V=800.0 PL=0
MOVL C00949 V=800.0 PL=0
MOVL C00950 V=800.0 PL=0
MOVL C00951 V=800.0 PL=0
MOVL C00952 V=800.0 PL=0
MOVL C00953 V=800.0 PL=0
MOVL C00954 V=800.0 PL=0
MOVL C00955 V=800.0 PL=0
MOVL C00956 V=800.0 PL=0
MOVL C00957 V=800.0 PL=0
MOVL C00958 V=800.0 PL=0
MOVL C00959 V=800.0 PL=0
MOVL C00960 V=800.0 PL=0
MOVL C00961 V=800.0 PL=0
MOVL C00962 V=800.0 PL=0
MOVL C00963 V=800.0 PL=0
MOVL C00964 V=800.0 PL=0
MOVL C00965 V=800.0 PL=0
MOVL C00966 V=800.0 PL=0
MOVL C00967 V=800.0 PL=0
MOVL C00968 V=800.0 PL=0
MOVL C00969 V=800.0 PL=0
MOVL C00970 V=800.0 PL=0
MOVL C00971 V=800.0 PL=0
MOVL C00972 V=800.0 PL=0
MOVL C00973 V=800.0 PL=0
MOVL C00974 V=800.0 PL=0
MOVL C00975 V=800.0 PL=0
MOVL C00976 V=800.0 PL=0
MOVL C00977 V=800.0 PL=0
MOVL C00978 V=800.0 PL=0
MOVL C00979 V=800.0 PL=0
MOVL C00980 V=800.0 PL=0
MOVL C00981 V=800.0 PL=0
MOVL C00982 V=800.0 PL=0
MOVL C00983 V=800.0 PL=0
MOVL C00984 V=800.0 PL=0
MOVL C00985 V=800.0 PL=0
MOVL C00986 V=800.0 PL=0
MOVL C00987 V=800.0 PL=0
MOVL C00988 V=800.0 PL=0
MOVL C00989 V=800.0 PL=0
MOVL C00990 V=800.0 PL=0
MOVL C00991 V=800.0 PL=0
MOVL C00992 V=800.0 PL=0
MOVL C00993 V=800.0 PL=0
MOVL C00994 V=800.0 PL=0
MOVL C00995 V=800.0 PL=0
MOVL C00996 V=800.0 PL=0
MOVL C00997 V=800.0 PL=0
MOVL C00998 V=800.0 PL=0
MOVL C00999 V=800.0 PL=0
MOVL C01000 V=800.0 PL=0
MOVL C01001 V=800.0 PL=0
MOVL C01002 V=800.0 PL=0
MOVL C01003 V=800.0 PL=0
MOVL C01004 V=800.0 PL=0
MOVL C01005 V=800.0 PL=0
MOVL C01006 V=800.0 PL=0
MOVL C01007 V=800.0 PL=0
MOVL C01008 V=800.0 PL=0
MOVL C01009 V=800.0 PL=0
MOVL C01010 V=800.0 PL=0
MOVL C01011 V=800.0 PL=0
MOVL C01012 V=800.0 PL=0
MOVL C01013 V=800.0 PL=0
MOVL C01014 V=800.0 PL=0
MOVL C01015 V=800.0 PL=0
MOVL C01016 V=800.0 PL=0
MOVL C01017 V=800.0 PL=0
MOVL C01018 V=800.0 PL=0
MOVL C01019 V=800.0 PL=0
MOVL C01020 V=800.0 PL=0
MOVL C01021 V=800.0 PL=0
MOVL C01022 V=800.0 PL=0
MOVL C01023 V=800.0 PL=0
MOVL C01024 V=800.0 PL=0
MOVL C01025 V=800.0 PL=0
MOVL C01026 V=800.0 PL=0
MOVL C01027 V=800.0 PL=0
MOVL C01028 V=800.0 PL=0
MOVL C01029 V=800.0 PL=0
MOVL C01030 V=800.0 PL=0
MOVL C01031 V=800.0 PL=0
MOVL C01032 V=800.0 PL=0
MOVL C01033 V=800.0 PL=0
MOVL C01034 V=800.0 PL=0
MOVL C01035 V=800.0 PL=0
MOVL C01036 V=800.0 PL=0
MOVL C01037 V=800.0 PL=0
MOVL C01038 V=800.0 PL=0
MOVL C01039 V=800.0 PL=0
MOVL C01040 V=800.0 PL=0
MOVL C01041 V=800.0 PL=0
MOVL C01042 V=800.0 PL=0
MOVL C01043 V=800.0 PL=0
MOVL C01044 V=800.0 PL=0
MOVL C01045 V=800.0 PL=0
MOVL C01046 V=800.0 PL=0
MOVL C01047 V=800.0 PL=0
MOVL C01048 V=800.0 PL=0
MOVL C01049 V=800.0 PL=0
MOVL C01050 V=800.0 PL=0
MOVL C01051 V=800.0 PL=0
MOVL C01052 V=800.0 PL=0
MOVL C01053 V=800.0 PL=0
MOVL C01054 V=800.0 PL=0
MOVL C01055 V=800.0 PL=0
MOVL C01056 V=800.0 PL=0
MOVL C01057 V=800.0 PL=0
MOVL C01058 V=800.0 PL=0
MOVL C01059 V=800.0 PL=0
MOVL C01060 V=800.0 PL=0
MOVL C01061 V=800.0 PL=0
MOVL C01062 V=800.0 PL=0
MOVL C01063 V=800.0 PL=0
MOVL C01064 V=800.0 PL=0
MOVL C01065 V=800.0 PL=0
MOVL C01066 V=800.0 PL=0
MOVL C01067 V=800.0 PL=0
MOVL C01068 V=800.0 PL=0
MOVL C01069 V=800.0 PL=0
MOVL C01070 V=800.0 PL=0
MOVL C01071 V=800.0 PL=0
MOVL C01072 V=800.0 PL=0
MOVL C01073 V=800.0 PL=0
MOVL C01074 V=800.0 PL=0
MOVL C01075 V=800.0 PL=0
MOVL C01076 V=800.0 PL=0
MOVL C01077 V=800.0 PL=0
MOVL C01078 V=800.0 PL=0
MOVL C01079 V=800.0 PL=0
MOVL C01080 V=800.0 PL=0
MOVL C01081 V=800.0 PL=0
MOVL C01082 V=800.0 PL=0
MOVL C01083 V=800.0 PL=0
MOVL C01084 V=800.0 PL=0
MOVL C01085 V=800.0 PL=0
MOVL C01086 V=800.0 PL=0
MOVL C01087 V=800.0 PL=0
MOVL C01088 V=800.0 PL=0
MOVL C01089 V=800.0 PL=0
MOVL C01090 V=800.0 PL=0
MOVL C01091 V=800.0 PL=0
MOVL C01092 V=800.0 PL=0
MOVL C01093 V=800.0 PL=0
MOVL C01094 V=800.0 PL=0
MOVL C01095 V=800.0 PL=0
MOVL C01096 V=800.0 PL=0
MOVL C01097 V=800.0 PL=0
MOVL C01098 V=800.0 PL=0
MOVL C01099 V=800.0 PL=0
MOVL C01100 V=800.0 PL=0
MOVL C01101 V=800.0 PL=0
MOVL C01102 V=800.0 PL=0
MOVL C01103 V=800.0 PL=0
MOVL C01104 V=800.0 PL=0
MOVL C01105 V=800.0 PL=0
MOVL C01106 V=800.0 PL=0
MOVL C01107 V=800.0 PL=0
MOVL C01108 V=800.0 PL=0
MOVL C01109 V=800.0 PL=0
MOVL C01110 V=800.0 PL=0
MOVL C01111 V=800.0 PL=0
MOVL C01112 V=800.0 PL=0
MOVL C01113 V=800.0 PL=0
MOVL C01114 V=800.0 PL=0
MOVL C01115 V=800.0 PL=0
MOVL C01116 V=800.0 PL=0
MOVL C01117 V=800.0 PL=0
MOVL C01118 V=800.0 PL=0
MOVL C01119 V=800.0 PL=0
MOVL C01120 V=800.0 PL=0
MOVL C01121 V=800.0 PL=0
MOVL C01122 V=800.0 PL=0
MOVL C01123 V=800.0 PL=0
MOVL C01124 V=800.0 PL=0
MOVL C01125 V=800.0 PL=0
MOVL C01126 V=800.0 PL=0
MOVL C01127 V=800.0 PL=0
MOVL C01128 V=800.0 PL=0
MOVL C01129 V=800.0 PL=0
MOVL C01130 V=800.0 PL=0
MOVL C01131 V=800.0 PL=0
MOVL C01132 V=800.0 PL=0
MOVL C01133 V=800.0 PL=0
MOVL C01134 V=800.0 PL=0
MOVL C01135 V=800.0 PL=0
MOVL C01136 V=800.0 PL=0
MOVL C01137 V=800.0 PL=0
MOVL C01138 V=800.0 PL=0
MOVL C01139 V=800.0 PL=0
MOVL C01140 V=800.0 PL=0
MOVL C01141 V=800.0 PL=0
MOVL C01142 V=800.0 PL=0
MOVL C01143 V=800.0 PL=0
MOVL C01144 V=800.0 PL=0
MOVL C01145 V=800.0 PL=0
MOVL C01146 V=800.0 PL=0
MOVL C01147 V=800.0 PL=0
MOVL C01148 V=800.0 PL=0
MOVL C01149 V=800.0 PL=0
MOVL C01150 V=800.0 PL=0
MOVL C01151 V=800.0 PL=0
MOVL C01152 V=800.0 PL=0
MOVL C01153 V=800.0 PL=0
MOVL C01154 V=800.0 PL=0
MOVL C01155 V=800.0 PL=0
MOVL C01156 V=800.0 PL=0
MOVL C01157 V=800.0 PL=0
MOVL C01158 V=800.0 PL=0
MOVL C01159 V=800.0 PL=0
MOVL C01160 V=800.0 PL=0
MOVL C01161 V=800.0 PL=0
MOVL C01162 V=800.0 PL=0
MOVL C01163 V=800.0 PL=0
MOVL C01164 V=800.0 PL=0
MOVL C01165 V=800.0 PL=0
MOVL C01166 V=800.0 PL=0
MOVL C01167 V=800.0 PL=0
MOVL C01168 V=800.0 PL=0
MOVL C01169 V=800.0 PL=0
MOVL C01170 V=800.0 PL=0
MOVL C01171 V=800.0 PL=0
MOVL C01172 V=800.0 PL=0
MOVL C01173 V=800.0 PL=0
MOVL C01174 V=800.0 PL=0
MOVL C01175 V=800.0 PL=0
MOVL C01176 V=800.0 PL=0
MOVL C01177 V=800.0 PL=0
MOVL C01178 V=800.0 PL=0
MOVL C01179 V=800.0 PL=0
MOVL C01180 V=800.0 PL=0
MOVL C01181 V=800.0 PL=0
MOVL C01182 V=800.0 PL=0
MOVL C01183 V=800.0 PL=0
MOVL C01184 V=800.0 PL=0
MOVL C01185 V=800.0 PL=0
MOVL C01186 V=800.0 PL=0
MOVL C01187 V=800.0 PL=0
MOVL C01188 V=800.0 PL=0
MOVL C01189 V=800.0 PL=0
MOVL C01190 V=800.0 PL=0
MOVL C01191 V=800.0 PL=0
MOVL C01192 V=800.0 PL=0
MOVL C01193 V=800.0 PL=0
MOVL C01194 V=800.0 PL=0
MOVL C01195 V=800.0 PL=0
MOVL C01196 V=800.0 PL=0
MOVL C01197 V=800.0 PL=0
MOVL C01198 V=800.0 PL=0
MOVL C01199 V=800.0 PL=0
MOVL C01200 V=800.0 PL=0
MOVL C01201 V=800.0 PL=0
MOVL C01202 V=800.0 PL=0
MOVL C01203 V=800.0 PL=0
MOVL C01204 V=800.0 PL=0
MOVL C01205 V=800.0 PL=0
MOVL C01206 V=800.0 PL=0
MOVL C01207 V=800.0 PL=0
MOVL C01208 V=800.0 PL=0
MOVL C01209 V=800.0 PL=0
MOVL C01210 V=800.0 PL=0
MOVL C01211 V=800.0 PL=0
MOVL C01212 V=800.0 PL=0
MOVL C01213 V=800.0 PL=0
MOVL C01214 V=800.0 PL=0
MOVL C01215 V=800.0 PL=0
MOVL C01216 V=800.0 PL=0
MOVL C01217 V=800.0 PL=0
MOVL C01218 V=800.0 PL=0
MOVL C01219 V=800.0 PL=0
MOVL C01220 V=800.0 PL=0
MOVL C01221 V=800.0 PL=0
MOVL C01222 V=800.0 PL=0
MOVL C01223 V=800.0 PL=0
MOVL C01224 V=800.0 PL=0
MOVL C01225 V=800.0 PL=0
MOVL C01226 V=800.0 PL=0
MOVL C01227 V=800.0 PL=0
MOVL C01228 V=800.0 PL=0
MOVL C01229 V=800.0 PL=0
MOVL C01230 V=800.0 PL=0
MOVL C01231 V=800.0 PL=0
MOVL C01232 V=800.0 PL=0
MOVL C01233 V=800.0 PL=0
MOVL C01234 V=800.0 PL=0
MOVL C01235 V=800.0 PL=0
MOVL C01236 V=800.0 PL=0
MOVL C01237 V=800.0 PL=0
MOVL C01238 V=800.0 PL=0
MOVL C01239 V=800.0 PL=0
MOVL C01240 V=800.0 PL=0
MOVL C01241 V=800.0 PL=0
MOVL C01242 V=800.0 PL=0
MOVL C01243 V=800.0 PL=0
MOVL C01244 V=800.0 PL=0
MOVL C01245 V=800.0 PL=0
MOVL C01246 V=800.0 PL=0
MOVL C01247 V=800.0 PL=0
MOVL C01248 V=800.0 PL=0
MOVL C01249 V=800.0 PL=0
MOVL C01250 V=800.0 PL=0
MOVL C01251 V=800.0 PL=0
MOVL C01252 V=800.0 PL=0
MOVL C01253 V=800.0 PL=0
MOVL C01254 V=800.0 PL=0
MOVL C01255 V=800.0 PL=0
MOVL C01256 V=800.0 PL=0
MOVL C01257 V=800.0 PL=0
MOVL C01258 V=800.0 PL=0
MOVL C01259 V=800.0 PL=0
MOVL C01260 V=800.0 PL=0
MOVL C01261 V=800.0 PL=0
MOVL C01262 V=800.0 PL=0
MOVL C01263 V=800.0 PL=0
MOVL C01264 V=800.0 PL=0
MOVL C01265 V=800.0 PL=0
MOVL C01266 V=800.0 PL=0
MOVL C01267 V=800.0 PL=0
MOVL C01268 V=800.0 PL=0
MOVL C01269 V=800.0 PL=0
MOVL C01270 V=800.0 PL=0
MOVL C01271 V=800.0 PL=0
MOVL C01272 V=800.0 PL=0
MOVL C01273 V=800.0 PL=0
MOVL C01274 V=800.0 PL=0
MOVL C01275 V=800.0 PL=0
MOVL C01276 V=800.0 PL=0
MOVL C01277 V=800.0 PL=0
MOVL C01278 V=800.0 PL=0
MOVL C01279 V=800.0 PL=0
MOVL C01280 V=800.0 PL=0
MOVL C01281 V=800.0 PL=0
MOVL C01282 V=800.0 PL=0
MOVL C01283 V=800.0 PL=0
MOVL C01284 V=800.0 PL=0
MOVL C01285 V=800.0 PL=0
MOVL C01286 V=800.0 PL=0
MOVL C01287 V=800.0 PL=0
MOVL C01288 V=800.0 PL=0
MOVL C01289 V=800.0 PL=0
MOVL C01290 V=800.0 PL=0
MOVL C01291 V=800.0 PL=0
MOVL C01292 V=800.0 PL=0
MOVL C01293 V=800.0 PL=0
MOVL C01294 V=800.0 PL=0
MOVL C01295 V=800.0 PL=0
MOVL C01296 V=800.0 PL=0
MOVL C01297 V=800.0 PL=0
MOVL C01298 V=800.0 PL=0
MOVL C01299 V=800.0 PL=0
MOVL C01300 V=800.0 PL=0
MOVL C01301 V=800.0 PL=0
MOVL C01302 V=800.0 PL=0
MOVL C01303 V=800.0 PL=0
MOVL C01304 V=800.0 PL=0
MOVL C01305 V=800.0 PL=0
MOVL C01306 V=800.0 PL=0
MOVL C01307 V=800.0 PL=0
MOVL C01308 V=800.0 PL=0
MOVL C01309 V=800.0 PL=0
MOVL C01310 V=800.0 PL=0
MOVL C01311 V=800.0 PL=0
MOVL C01312 V=800.0 PL=0
MOVL C01313 V=800.0 PL=0
MOVL C01314 V=800.0 PL=0
MOVL C01315 V=800.0 PL=0
MOVL C01316 V=800.0 PL=0
MOVL C01317 V=800.0 PL=0
MOVL C01318 V=800.0 PL=0
MOVL C01319 V=800.0 PL=0
MOVL C01320 V=800.0 PL=0
MOVL C01321 V=800.0 PL=0
MOVL C01322 V=800.0 PL=0
MOVL C01323 V=800.0 PL=0
MOVL C01324 V=800.0 PL=0
MOVL C01325 V=800.0 PL=0
MOVL C01326 V=800.0 PL=0
MOVL C01327 V=800.0 PL=0
MOVL C01328 V=800.0 PL=0
MOVL C01329 V=800.0 PL=0
MOVL C01330 V=800.0 PL=0
MOVL C01331 V=800.0 PL=0
MOVL C01332 V=800.0 PL=0
MOVL C01333 V=800.0 PL=0
MOVL C01334 V=800.0 PL=0
MOVL C01335 V=800.0 PL=0
MOVL C01336 V=800.0 PL=0
MOVL C01337 V=800.0 PL=0
MOVL C01338 V=800.0 PL=0
MOVL C01339 V=800.0 PL=0
MOVL C01340 V=800.0 PL=0
MOVL C01341 V=800.0 PL=0
MOVL C01342 V=800.0 PL=0
MOVL C01343 V=800.0 PL=0
MOVL C01344 V=800.0 PL=0
MOVL C01345 V=800.0 PL=0
MOVL C01346 V=800.0 PL=0
MOVL C01347 V=800.0 PL=0
MOVL C01348 V=800.0 PL=0
MOVL C01349 V=800.0 PL=0
MOVL C01350 V=800.0 PL=0
MOVL C01351 V=800.0 PL=0
MOVL C01352 V=800.0 PL=0
MOVL C01353 V=800.0 PL=0
MOVL C01354 V=800.0 PL=0
MOVL C01355 V=800.0 PL=0
MOVL C01356 V=800.0 PL=0
MOVL C01357 V=800.0 PL=0
MOVL C01358 V=800.0 PL=0
MOVL C01359 V=800.0 PL=0
MOVL C01360 V=800.0 PL=0
MOVL C01361 V=800.0 PL=0
MOVL C01362 V=800.0 PL=0
MOVL C01363 V=800.0 PL=0
MOVL C01364 V=800.0 PL=0
MOVL C01365 V=800.0 PL=0
MOVL C01366 V=800.0 PL=0
MOVL C01367 V=800.0 PL=0
MOVL C01368 V=800.0 PL=0
MOVL C01369 V=800.0 PL=0
MOVL C01370 V=800.0 PL=0
MOVL C01371 V=800.0 PL=0
MOVL C01372 V=800.0 PL=0
MOVL C01373 V=800.0 PL=0
MOVL C01374 V=800.0 PL=0
MOVL C01375 V=800.0 PL=0
MOVL C01376 V=800.0 PL=0
MOVL C01377 V=800.0 PL=0
MOVL C01378 V=800.0 PL=0
MOVL C01379 V=800.0 PL=0
MOVL C01380 V=800.0 PL=0
MOVL C01381 V=800.0 PL=0
MOVL C01382 V=800.0 PL=0
MOVL C01383 V=800.0 PL=0
MOVL C01384 V=800.0 PL=0
MOVL C01385 V=800.0 PL=0
MOVL C01386 V=800.0 PL=0
MOVL C01387 V=800.0 PL=0
MOVL C01388 V=800.0 PL=0
MOVL C01389 V=800.0 PL=0
MOVL C01390 V=800.0 PL=0
MOVL C01391 V=800.0 PL=0
MOVL C01392 V=800.0 PL=0
MOVL C01393 V=800.0 PL=0
MOVL C01394 V=800.0 PL=0
MOVL C01395 V=800.0 PL=0
MOVL C01396 V=800.0 PL=0
MOVL C01397 V=800.0 PL=0
MOVL C01398 V=800.0 PL=0
MOVL C01399 V=800.0 PL=0
MOVL C01400 V=800.0 PL=0
MOVL C01401 V=800.0 PL=0
MOVL C01402 V=800.0 PL=0
MOVL C01403 V=800.0 PL=0
MOVL C01404 V=800.0 PL=0
MOVL C01405 V=800.0 PL=0
MOVL C01406 V=800.0 PL=0
MOVL C01407 V=800.0 PL=0
MOVL C01408 V=800.0 PL=0
MOVL C01409 V=800.0 PL=0
MOVL C01410 V=800.0 PL=0
MOVL C01411 V=800.0 PL=0
MOVL C01412 V=800.0 PL=0
MOVL C01413 V=800.0 PL=0
MOVL C01414 V=800.0 PL=0
MOVL C01415 V=800.0 PL=0
MOVL C01416 V=800.0 PL=0
MOVL C01417 V=800.0 PL=0
MOVL C01418 V=800.0 PL=0
MOVL C01419 V=800.0 PL=0
MOVL C01420 V=800.0 PL=0
MOVL C01421 V=800.0 PL=0
MOVL C01422 V=800.0 PL=0
MOVL C01423 V=800.0 PL=0
MOVL C01424 V=800.0 PL=0
MOVL C01425 V=800.0 PL=0
MOVL C01426 V=800.0 PL=0
MOVL C01427 V=800.0 PL=0
MOVL C01428 V=800.0 PL=0
MOVL C01429 V=800.0 PL=0
MOVL C01430 V=800.0 PL=0
MOVL C01431 V=800.0 PL=0
MOVL C01432 V=800.0 PL=0
MOVL C01433 V=800.0 PL=0
MOVL C01434 V=800.0 PL=0
MOVL C01435 V=800.0 PL=0
MOVL C01436 V=800.0 PL=0
MOVL C01437 V=800.0 PL=0
MOVL C01438 V=800.0 PL=0
MOVL C01439 V=800.0 PL=0
MOVL C01440 V=800.0 PL=0
MOVL C01441 V=800.0 PL=0
MOVL C01442 V=800.0 PL=0
MOVL C01443 V=800.0 PL=0
MOVL C01444 V=800.0 PL=0
MOVL C01445 V=800.0 PL=0
MOVL C01446 V=800.0 PL=0
MOVL C01447 V=800.0 PL=0
MOVL C01448 V=800.0 PL=0
MOVL C01449 V=800.0 PL=0
MOVL C01450 V=800.0 PL=0
MOVL C01451 V=800.0 PL=0
MOVL C01452 V=800.0 PL=0
MOVL C01453 V=800.0 PL=0
MOVL C01454 V=800.0 PL=0
MOVL C01455 V=800.0 PL=0
MOVL C01456 V=800.0 PL=0
MOVL C01457 V=800.0 PL=0
MOVL C01458 V=800.0 PL=0
MOVL C01459 V=800.0 PL=0
MOVL C01460 V=800.0 PL=0
MOVL C01461 V=800.0 PL=0
MOVL C01462 V=800.0 PL=0
MOVL C01463 V=800.0 PL=0
MOVL C01464 V=800.0 PL=0
MOVL C01465 V=800.0 PL=0
MOVL C01466 V=800.0 PL=0
MOVL C01467 V=800.0 PL=0
MOVL C01468 V=800.0 PL=0
MOVL C01469 V=800.0 PL=0
MOVL C01470 V=800.0 PL=0
MOVL C01471 V=800.0 PL=0
MOVL C01472 V=800.0 PL=0
MOVL C01473 V=800.0 PL=0
MOVL C01474 V=800.0 PL=0
MOVL C01475 V=800.0 PL=0
MOVL C01476 V=800.0 PL=0
MOVL C01477 V=800.0 PL=0
MOVL C01478 V=800.0 PL=0
MOVL C01479 V=800.0 PL=0
MOVL C01480 V=800.0 PL=0
MOVL C01481 V=800.0 PL=0
MOVL C01482 V=800.0 PL=0
MOVL C01483 V=800.0 PL=0
MOVL C01484 V=800.0 PL=0
MOVL C01485 V=800.0 PL=0
MOVL C01486 V=800.0 PL=0
MOVL C01487 V=800.0 PL=0
MOVL C01488 V=800.0 PL=0
MOVL C01489 V=800.0 PL=0
MOVL C01490 V=800.0 PL=0
MOVL C01491 V=800.0 PL=0
MOVL C01492 V=800.0 PL=0
MOVL C01493 V=800.0 PL=0
MOVL C01494 V=800.0 PL=0
MOVL C01495 V=800.0 PL=0
MOVL C01496 V=800.0 PL=0
MOVL C01497 V=800.0 PL=0
MOVL C01498 V=800.0 PL=0
MOVL C01499 V=800.0 PL=0
MOVL C01500 V=800.0 PL=0
MOVL C01501 V=800.0 PL=0
MOVL C01502 V=800.0 PL=0
MOVL C01503 V=800.0 PL=0
MOVL C01504 V=800.0 PL=0
MOVL C01505 V=800.0 PL=0
MOVL C01506 V=800.0 PL=0
MOVL C01507 V=800.0 PL=0
MOVL C01508 V=800.0 PL=0
MOVL C01509 V=800.0 PL=0
MOVL C01510 V=800.0 PL=0
MOVL C01511 V=800.0 PL=0
MOVL C01512 V=800.0 PL=0
MOVL C01513 V=800.0 PL=0
MOVL C01514 V=800.0 PL=0
MOVL C01515 V=800.0 PL=0
MOVL C01516 V=800.0 PL=0
MOVL C01517 V=800.0 PL=0
MOVL C01518 V=800.0 PL=0
MOVL C01519 V=800.0 PL=0
MOVL C01520 V=800.0 PL=0
MOVL C01521 V=800.0 PL=0
MOVL C01522 V=800.0 PL=0
MOVL C01523 V=800.0 PL=0
MOVL C01524 V=800.0 PL=0
MOVL C01525 V=800.0 PL=0
MOVL C01526 V=800.0 PL=0
MOVL C01527 V=800.0 PL=0
MOVL C01528 V=800.0 PL=0
MOVL C01529 V=800.0 PL=0
MOVL C01530 V=800.0 PL=0
MOVL C01531 V=800.0 PL=0
MOVL C01532 V=800.0 PL=0
MOVL C01533 V=800.0 PL=0
MOVL C01534 V=800.0 PL=0
MOVL C01535 V=800.0 PL=0
MOVL C01536 V=800.0 PL=0
MOVL C01537 V=800.0 PL=0
MOVL C01538 V=800.0 PL=0
MOVL C01539 V=800.0 PL=0
MOVL C01540 V=800.0 PL=0
MOVL C01541 V=800.0 PL=0
MOVL C01542 V=800.0 PL=0
MOVL C01543 V=800.0 PL=0
MOVL C01544 V=800.0 PL=0
MOVL C01545 V=800.0 PL=0
MOVL C01546 V=800.0 PL=0
MOVL C01547 V=800.0 PL=0
MOVL C01548 V=800.0 PL=0
MOVL C01549 V=800.0 PL=0
MOVL C01550 V=800.0 PL=0
MOVL C01551 V=800.0 PL=0
MOVL C01552 V=800.0 PL=0
MOVL C01553 V=800.0 PL=0
MOVL C01554 V=800.0 PL=0
MOVL C01555 V=800.0 PL=0
MOVL C01556 V=800.0 PL=0
MOVL C01557 V=800.0 PL=0
MOVL C01558 V=800.0 PL=0
MOVL C01559 V=800.0 PL=0
MOVL C01560 V=800.0 PL=0
MOVL C01561 V=800.0 PL=0
MOVL C01562 V=800.0 PL=0
MOVL C01563 V=800.0 PL=0
MOVL C01564 V=800.0 PL=0
MOVL C01565 V=800.0 PL=0
MOVL C01566 V=800.0 PL=0
MOVL C01567 V=800.0 PL=0
MOVL C01568 V=800.0 PL=0
MOVL C01569 V=800.0 PL=0
MOVL C01570 V=800.0 PL=0
MOVL C01571 V=800.0 PL=0
MOVL C01572 V=800.0 PL=0
MOVL C01573 V=800.0 PL=0
MOVL C01574 V=800.0 PL=0
MOVL C01575 V=800.0 PL=0
MOVL C01576 V=800.0 PL=0
MOVL C01577 V=800.0 PL=0
MOVL C01578 V=800.0 PL=0
MOVL C01579 V=800.0 PL=0
MOVL C01580 V=800.0 PL=0
MOVL C01581 V=800.0 PL=0
MOVL C01582 V=800.0 PL=0
MOVL C01583 V=800.0 PL=0
MOVL C01584 V=800.0 PL=0
MOVL C01585 V=800.0 PL=0
MOVL C01586 V=800.0 PL=0
MOVL C01587 V=800.0 PL=0
MOVL C01588 V=800.0 PL=0
MOVL C01589 V=800.0 PL=0
MOVL C01590 V=800.0 PL=0
MOVL C01591 V=800.0 PL=0
MOVL C01592 V=800.0 PL=0
MOVL C01593 V=800.0 PL=0
MOVL C01594 V=800.0 PL=0
MOVL C01595 V=800.0 PL=0
MOVL C01596 V=800.0 PL=0
MOVL C01597 V=800.0 PL=0
MOVL C01598 V=800.0 PL=0
MOVL C01599 V=800.0 PL=0
MOVL C01600 V=800.0 PL=0
MOVL C01601 V=800.0 PL=0
MOVL C01602 V=800.0 PL=0
MOVL C01603 V=800.0 PL=0
MOVL C01604 V=800.0 PL=0
MOVL C01605 V=800.0 PL=0
MOVL C01606 V=800.0 PL=0
MOVL C01607 V=800.0 PL=0
MOVL C01608 V=800.0 PL=0
MOVL C01609 V=800.0 PL=0
MOVL C01610 V=800.0 PL=0
MOVL C01611 V=800.0 PL=0
MOVL C01612 V=800.0 PL=0
MOVL C01613 V=800.0 PL=0
MOVL C01614 V=800.0 PL=0
MOVL C01615 V=800.0 PL=0
MOVL C01616 V=800.0 PL=0
MOVL C01617 V=800.0 PL=0
MOVL C01618 V=800.0 PL=0
MOVL C01619 V=800.0 PL=0
MOVL C01620 V=800.0 PL=0
MOVL C01621 V=800.0 PL=0
MOVL C01622 V=800.0 PL=0
MOVL C01623 V=800.0 PL=0
MOVL C01624 V=800.0 PL=0
MOVL C01625 V=800.0 PL=0
MOVL C01626 V=800.0 PL=0
MOVL C01627 V=800.0 PL=0
MOVL C01628 V=800.0 PL=0
MOVL C01629 V=800.0 PL=0
MOVL C01630 V=800.0 PL=0
MOVL C01631 V=800.0 PL=0
MOVL C01632 V=800.0 PL=0
MOVL C01633 V=800.0 PL=0
MOVL C01634 V=800.0 PL=0
MOVL C01635 V=800.0 PL=0
MOVL C01636 V=800.0 PL=0
MOVL C01637 V=800.0 PL=0
MOVL C01638 V=800.0 PL=0
MOVL C01639 V=800.0 PL=0
MOVL C01640 V=800.0 PL=0
MOVL C01641 V=800.0 PL=0
MOVL C01642 V=800.0 PL=0
MOVL C01643 V=800.0 PL=0
MOVL C01644 V=800.0 PL=0
MOVL C01645 V=800.0 PL=0
MOVL C01646 V=800.0 PL=0
MOVL C01647 V=800.0 PL=0
MOVL C01648 V=800.0 PL=0
MOVL C01649 V=800.0 PL=0
MOVL C01650 V=800.0 PL=0
MOVL C01651 V=800.0 PL=0
MOVL C01652 V=800.0 PL=0
MOVL C01653 V=800.0 PL=0
MOVL C01654 V=800.0 PL=0
MOVL C01655 V=800.0 PL=0
MOVL C01656 V=800.0 PL=0
MOVL C01657 V=800.0 PL=0
MOVL C01658 V=800.0 PL=0
MOVL C01659 V=800.0 PL=0
MOVL C01660 V=800.0 PL=0
MOVL C01661 V=800.0 PL=0
MOVL C01662 V=800.0 PL=0
MOVL C01663 V=800.0 PL=0
MOVL C01664 V=800.0 PL=0
MOVL C01665 V=800.0 PL=0
MOVL C01666 V=800.0 PL=0
MOVL C01667 V=800.0 PL=0
MOVL C01668 V=800.0 PL=0
MOVL C01669 V=800.0 PL=0
MOVL C01670 V=800.0 PL=0
MOVL C01671 V=800.0 PL=0
MOVL C01672 V=800.0 PL=0
MOVL C01673 V=800.0 PL=0
MOVL C01674 V=800.0 PL=0
MOVL C01675 V=800.0 PL=0
MOVL C01676 V=800.0 PL=0
MOVL C01677 V=800.0 PL=0
MOVL C01678 V=800.0 PL=0
MOVL C01679 V=800.0 PL=0
MOVL C01680 V=800.0 PL=0
MOVL C01681 V=800.0 PL=0
MOVL C01682 V=800.0 PL=0
MOVL C01683 V=800.0 PL=0
MOVL C01684 V=800.0 PL=0
MOVL C01685 V=800.0 PL=0
MOVL C01686 V=800.0 PL=0
MOVL C01687 V=800.0 PL=0
MOVL C01688 V=800.0 PL=0
MOVL C01689 V=800.0 PL=0
MOVL C01690 V=800.0 PL=0
MOVL C01691 V=800.0 PL=0
MOVL C01692 V=800.0 PL=0
MOVL C01693 V=800.0 PL=0
MOVL C01694 V=800.0 PL=0
MOVL C01695 V=800.0 PL=0
MOVL C01696 V=800.0 PL=0
MOVL C01697 V=800.0 PL=0
MOVL C01698 V=800.0 PL=0
MOVL C01699 V=800.0 PL=0
MOVL C01700 V=800.0 PL=0
MOVL C01701 V=800.0 PL=0
MOVL C01702 V=800.0 PL=0
MOVL C01703 V=800.0 PL=0
MOVL C01704 V=800.0 PL=0
MOVL C01705 V=800.0 PL=0
MOVL C01706 V=800.0 PL=0
MOVL C01707 V=800.0 PL=0
MOVL C01708 V=800.0 PL=0
MOVL C01709 V=800.0 PL=0
MOVL C01710 V=800.0 PL=0
MOVL C01711 V=800.0 PL=0
MOVL C01712 V=800.0 PL=0
MOVL C01713 V=800.0 PL=0
MOVL C01714 V=800.0 PL=0
MOVL C01715 V=800.0 PL=0
MOVL C01716 V=800.0 PL=0
MOVL C01717 V=800.0 PL=0
MOVL C01718 V=800.0 PL=0
MOVL C01719 V=800.0 PL=0
MOVL C01720 V=800.0 PL=0
MOVL C01721 V=800.0 PL=0
MOVL C01722 V=800.0 PL=0
MOVL C01723 V=800.0 PL=0
MOVL C01724 V=800.0 PL=0
MOVL C01725 V=800.0 PL=0
MOVL C01726 V=800.0 PL=0
MOVL C01727 V=800.0 PL=0
MOVL C01728 V=800.0 PL=0
MOVL C01729 V=800.0 PL=0
MOVL C01730 V=800.0 PL=0
MOVL C01731 V=800.0 PL=0
MOVL C01732 V=800.0 PL=0
MOVL C01733 V=800.0 PL=0
MOVL C01734 V=800.0 PL=0
MOVL C01735 V=800.0 PL=0
MOVL C01736 V=800.0 PL=0
MOVL C01737 V=800.0 PL=0
MOVL C01738 V=800.0 PL=0
MOVL C01739 V=800.0 PL=0
MOVL C01740 V=800.0 PL=0
MOVL C01741 V=800.0 PL=0
MOVL C01742 V=800.0 PL=0
MOVL C01743 V=800.0 PL=0
MOVL C01744 V=800.0 PL=0
MOVL C01745 V=800.0 PL=0
MOVL C01746 V=800.0 PL=0
MOVL C01747 V=800.0 PL=0
MOVL C01748 V=800.0 PL=0
MOVL C01749 V=800.0 PL=0
MOVL C01750 V=800.0 PL=0
MOVL C01751 V=800.0 PL=0
MOVL C01752 V=800.0 PL=0
MOVL C01753 V=800.0 PL=0
MOVL C01754 V=800.0 PL=0
MOVL C01755 V=800.0 PL=0
MOVL C01756 V=800.0 PL=0
MOVL C01757 V=800.0 PL=0
MOVL C01758 V=800.0 PL=0
MOVL C01759 V=800.0 PL=0
MOVL C01760 V=800.0 PL=0
MOVL C01761 V=800.0 PL=0
MOVL C01762 V=800.0 PL=0
MOVL C01763 V=800.0 PL=0
MOVL C01764 V=800.0 PL=0
MOVL C01765 V=800.0 PL=0
MOVL C01766 V=800.0 PL=0
MOVL C01767 V=800.0 PL=0
MOVL C01768 V=800.0 PL=0
MOVL C01769 V=800.0 PL=0
MOVL C01770 V=800.0 PL=0
MOVL C01771 V=800.0 PL=0
MOVL C01772 V=800.0 PL=0
MOVL C01773 V=800.0 PL=0
MOVL C01774 V=800.0 PL=0
MOVL C01775 V=800.0 PL=0
MOVL C01776 V=800.0 PL=0
MOVL C01777 V=800.0 PL=0
MOVL C01778 V=800.0 PL=0
MOVL C01779 V=800.0 PL=0
MOVL C01780 V=800.0 PL=0
MOVL C01781 V=800.0 PL=0
MOVL C01782 V=800.0 PL=0
MOVL C01783 V=800.0 PL=0
MOVL C01784 V=800.0 PL=0
MOVL C01785 V=800.0 PL=0
MOVL C01786 V=800.0 PL=0
MOVL C01787 V=800.0 PL=0
MOVL C01788 V=800.0 PL=0
MOVL C01789 V=800.0 PL=0
MOVL C01790 V=800.0 PL=0
MOVL C01791 V=800.0 PL=0
MOVL C01792 V=800.0 PL=0
MOVL C01793 V=800.0 PL=0
MOVL C01794 V=800.0 PL=0
MOVL C01795 V=800.0 PL=0
MOVL C01796 V=800.0 PL=0
MOVL C01797 V=800.0 PL=0
MOVL C01798 V=800.0 PL=0
MOVL C01799 V=800.0 PL=0
MOVL C01800 V=800.0 PL=0
MOVL C01801 V=800.0 PL=0
MOVL C01802 V=800.0 PL=0
MOVL C01803 V=800.0 PL=0
MOVL C01804 V=800.0 PL=0
MOVL C01805 V=800.0 PL=0
MOVL C01806 V=800.0 PL=0
MOVL C01807 V=800.0 PL=0
MOVL C01808 V=800.0 PL=0
MOVL C01809 V=800.0 PL=0
MOVL C01810 V=800.0 PL=0
MOVL C01811 V=800.0 PL=0
MOVL C01812 V=800.0 PL=0
MOVL C01813 V=800.0 PL=0
MOVL C01814 V=800.0 PL=0
MOVL C01815 V=800.0 PL=0
MOVL C01816 V=800.0 PL=0
MOVL C01817 V=800.0 PL=0
MOVL C01818 V=800.0 PL=0
MOVL C01819 V=800.0 PL=0
MOVL C01820 V=800.0 PL=0
MOVL C01821 V=800.0 PL=0
MOVL C01822 V=800.0 PL=0
MOVL C01823 V=800.0 PL=0
MOVL C01824 V=800.0 PL=0
MOVL C01825 V=800.0 PL=0
MOVL C01826 V=800.0 PL=0
MOVL C01827 V=800.0 PL=0
MOVL C01828 V=800.0 PL=0
MOVL C01829 V=800.0 PL=0
MOVL C01830 V=800.0 PL=0
MOVL C01831 V=800.0 PL=0
MOVL C01832 V=800.0 PL=0
MOVL C01833 V=800.0 PL=0
MOVL C01834 V=800.0 PL=0
MOVL C01835 V=800.0 PL=0
MOVL C01836 V=800.0 PL=0
MOVL C01837 V=800.0 PL=0
MOVL C01838 V=800.0 PL=0
MOVL C01839 V=800.0 PL=0
MOVL C01840 V=800.0 PL=0
MOVL C01841 V=800.0 PL=0
MOVL C01842 V=800.0 PL=0
MOVL C01843 V=800.0 PL=0
MOVL C01844 V=800.0 PL=0
MOVL C01845 V=800.0 PL=0
MOVL C01846 V=800.0 PL=0
MOVL C01847 V=800.0 PL=0
MOVL C01848 V=800.0 PL=0
MOVL C01849 V=800.0 PL=0
MOVL C01850 V=800.0 PL=0
MOVL C01851 V=800.0 PL=0
MOVL C01852 V=800.0 PL=0
MOVL C01853 V=800.0 PL=0
MOVL C01854 V=800.0 PL=0
MOVL C01855 V=800.0 PL=0
MOVL C01856 V=800.0 PL=0
MOVL C01857 V=800.0 PL=0
MOVL C01858 V=800.0 PL=0
MOVL C01859 V=800.0 PL=0
MOVL C01860 V=800.0 PL=0
MOVL C01861 V=800.0 PL=0
MOVL C01862 V=800.0 PL=0
MOVL C01863 V=800.0 PL=0
MOVL C01864 V=800.0 PL=0
MOVL C01865 V=800.0 PL=0
MOVL C01866 V=800.0 PL=0
MOVL C01867 V=800.0 PL=0
MOVL C01868 V=800.0 PL=0
MOVL C01869 V=800.0 PL=0
MOVL C01870 V=800.0 PL=0
MOVL C01871 V=800.0 PL=0
MOVL C01872 V=800.0 PL=0
MOVL C01873 V=800.0 PL=0
MOVL C01874 V=800.0 PL=0
MOVL C01875 V=800.0 PL=0
MOVL C01876 V=800.0 PL=0
MOVL C01877 V=800.0 PL=0
MOVL C01878 V=800.0 PL=0
MOVL C01879 V=800.0 PL=0
MOVL C01880 V=800.0 PL=0
MOVL C01881 V=800.0 PL=0
MOVL C01882 V=800.0 PL=0
MOVL C01883 V=800.0 PL=0
MOVL C01884 V=800.0 PL=0
MOVL C01885 V=800.0 PL=0
MOVL C01886 V=800.0 PL=0
MOVL C01887 V=800.0 PL=0
MOVL C01888 V=800.0 PL=0
MOVL C01889 V=800.0 PL=0
MOVL C01890 V=800.0 PL=0
MOVL C01891 V=800.0 PL=0
MOVL C01892 V=800.0 PL=0
MOVL C01893 V=800.0 PL=0
MOVL C01894 V=800.0 PL=0
MOVL C01895 V=800.0 PL=0
MOVL C01896 V=800.0 PL=0
MOVL C01897 V=800.0 PL=0
MOVL C01898 V=800.0 PL=0
MOVL C01899 V=800.0 PL=0
MOVL C01900 V=800.0 PL=0
MOVL C01901 V=800.0 PL=0
MOVL C01902 V=800.0 PL=0
MOVL C01903 V=800.0 PL=0
MOVL C01904 V=800.0 PL=0
MOVL C01905 V=800.0 PL=0
MOVL C01906 V=800.0 PL=0
MOVL C01907 V=800.0 PL=0
MOVL C01908 V=800.0 PL=0
MOVL C01909 V=800.0 PL=0
MOVL C01910 V=800.0 PL=0
MOVL C01911 V=800.0 PL=0
MOVL C01912 V=800.0 PL=0
MOVL C01913 V=800.0 PL=0
MOVL C01914 V=800.0 PL=0
MOVL C01915 V=800.0 PL=0
MOVL C01916 V=800.0 PL=0
MOVL C01917 V=800.0 PL=0
MOVL C01918 V=800.0 PL=0
MOVL C01919 V=800.0 PL=0
MOVL C01920 V=800.0 PL=0
MOVL C01921 V=800.0 PL=0
MOVL C01922 V=800.0 PL=0
MOVL C01923 V=800.0 PL=0
MOVL C01924 V=800.0 PL=0
MOVL C01925 V=800.0 PL=0
MOVL C01926 V=800.0 PL=0
MOVL C01927 V=800.0 PL=0
MOVL C01928 V=800.0 PL=0
MOVL C01929 V=800.0 PL=0
MOVL C01930 V=800.0 PL=0
MOVL C01931 V=800.0 PL=0
MOVL C01932 V=800.0 PL=0
MOVL C01933 V=800.0 PL=0
MOVL C01934 V=800.0 PL=0
MOVL C01935 V=800.0 PL=0
MOVL C01936 V=800.0 PL=0
MOVL C01937 V=800.0 PL=0
MOVL C01938 V=800.0 PL=0
MOVL C01939 V=800.0 PL=0
MOVL C01940 V=800.0 PL=0
MOVL C01941 V=800.0 PL=0
MOVL C01942 V=800.0 PL=0
MOVL C01943 V=800.0 PL=0
MOVL C01944 V=800.0 PL=0
MOVL C01945 V=800.0 PL=0
MOVL C01946 V=800.0 PL=0
MOVL C01947 V=800.0 PL=0
MOVL C01948 V=800.0 PL=0
MOVL C01949 V=800.0 PL=0
MOVL C01950 V=800.0 PL=0
MOVL C01951 V=800.0 PL=0
MOVL C01952 V=800.0 PL=0
MOVL C01953 V=800.0 PL=0
MOVL C01954 V=800.0 PL=0
MOVL C01955 V=800.0 PL=0
MOVL C01956 V=800.0 PL=0
MOVL C01957 V=800.0 PL=0
MOVL C01958 V=800.0 PL=0
MOVL C01959 V=800.0 PL=0
MOVL C01960 V=800.0 PL=0
MOVL C01961 V=800.0 PL=0
MOVL C01962 V=800.0 PL=0
MOVL C01963 V=800.0 PL=0
MOVL C01964 V=800.0 PL=0
MOVL C01965 V=800.0 PL=0
MOVL C01966 V=800.0 PL=0
MOVL C01967 V=800.0 PL=0
MOVL C01968 V=800.0 PL=0
MOVL C01969 V=800.0 PL=0
MOVL C01970 V=800.0 PL=0
MOVL C01971 V=800.0 PL=0
MOVL C01972 V=800.0 PL=0
MOVL C01973 V=800.0 PL=0
MOVL C01974 V=800.0 PL=0
MOVL C01975 V=800.0 PL=0
MOVL C01976 V=800.0 PL=0
MOVL C01977 V=800.0 PL=0
MOVL C01978 V=800.0 PL=0
MOVL C01979 V=800.0 PL=0
MOVL C01980 V=800.0 PL=0
MOVL C01981 V=800.0 PL=0
MOVL C01982 V=800.0 PL=0
MOVL C01983 V=800.0 PL=0
MOVL C01984 V=800.0 PL=0
MOVL C01985 V=800.0 PL=0
MOVL C01986 V=800.0 PL=0
MOVL C01987 V=800.0 PL=0
MOVL C01988 V=800.0 PL=0
MOVL C01989 V=800.0 PL=0
MOVL C01990 V=800.0 PL=0
MOVL C01991 V=800.0 PL=0
MOVL C01992 V=800.0 PL=0
MOVL C01993 V=800.0 PL=0
MOVL C01994 V=800.0 PL=0
MOVL C01995 V=800.0 PL=0
MOVL C01996 V=800.0 PL=0
MOVL C01997 V=800.0 PL=0
MOVL C01998 V=800.0 PL=0
MOVL C01999 V=800.0 PL=0
MOVL C02000 V=800.0 PL=0
MOVL C02001 V=800.0 PL=0
MOVL C02002 V=800.0 PL=0
MOVL C02003 V=800.0 PL=0
MOVL C02004 V=800.0 PL=0
MOVL C02005 V=800.0 PL=0
MOVL C02006 V=800.0 PL=0
MOVL C02007 V=800.0 PL=0
MOVL C02008 V=800.0 PL=0
MOVL C02009 V=800.0 PL=0
MOVL C02010 V=800.0 PL=0
MOVL C02011 V=800.0 PL=0
MOVL C02012 V=800.0 PL=0
MOVL C02013 V=800.0 PL=0
MOVL C02014 V=800.0 PL=0
MOVL C02015 V=800.0 PL=0
MOVL C02016 V=800.0 PL=0
MOVL C02017 V=800.0 PL=0
MOVL C02018 V=800.0 PL=0
MOVL C02019 V=800.0 PL=0
MOVL C02020 V=800.0 PL=0
MOVL C02021 V=800.0 PL=0
MOVL C02022 V=800.0 PL=0
MOVL C02023 V=800.0 PL=0
MOVL C02024 V=800.0 PL=0
MOVL C02025 V=800.0 PL=0
MOVL C02026 V=800.0 PL=0
MOVL C02027 V=800.0 PL=0
MOVL C02028 V=800.0 PL=0
MOVL C02029 V=800.0 PL=0
MOVL C02030 V=800.0 PL=0
MOVL C02031 V=800.0 PL=0
MOVL C02032 V=800.0 PL=0
MOVL C02033 V=800.0 PL=0
MOVL C02034 V=800.0 PL=0
MOVL C02035 V=800.0 PL=0
MOVL C02036 V=800.0 PL=0
MOVL C02037 V=800.0 PL=0
MOVL C02038 V=800.0 PL=0
MOVL C02039 V=800.0 PL=0
MOVL C02040 V=800.0 PL=0
MOVL C02041 V=800.0 PL=0
